LIN {X -0.265,Y -656.677,Z 1261.343,A 0.000,B 0.000,C 90.000,E1 97.757} C_DIS
LIN {X -0.061,Y -653.194,Z 1261.340,A 0.000,B 0.000,C 90.000,E1 97.125} C_DIS
LIN {X 0.226,Y -650.001,Z 1261.337,A 0.000,B 0.000,C 90.000,E1 96.606} C_DIS
LIN {X -0.200,Y -645.461,Z 1261.333,A 0.000,B 0.000,C 90.000,E1 96.024} C_DIS
LIN {X 0.088,Y -642.536,Z 1261.331,A 0.000,B 0.000,C 90.000,E1 95.625} C_DIS
LIN {X 0.172,Y -637.015,Z 1261.328,A 0.000,B 0.000,C 90.000,E1 94.992} C_DIS
LIN {X 0.261,Y -630.867,Z 1261.324,A 0.000,B 0.000,C 90.000,E1 94.359} C_DIS
LIN {X -0.014,Y -625.710,Z 1261.322,A 0.000,B 0.000,C 90.000,E1 93.898} C_DIS
LIN {X -0.161,Y -618.882,Z 1261.318,A 0.000,B 0.000,C 90.000,E1 93.326} C_DIS
LIN {X -0.104,Y -614.516,Z 1261.317,A 0.000,B 0.000,C 90.000,E1 92.980} C_DIS
LIN {X 0.202,Y -608.733,Z 1261.314,A 0.000,B 0.000,C 90.000,E1 92.522} C_DIS
LIN {X 0.170,Y -601.165,Z 1261.311,A 0.000,B 0.000,C 90.000,E1 92.007} C_DIS
LIN {X 0.030,Y -596.550,Z 1261.310,A 0.000,B 0.000,C 90.000,E1 91.718} C_DIS
LIN {X 0.285,Y -589.902,Z 1261.307,A 0.000,B 0.000,C 90.000,E1 91.318} C_DIS
LIN {X -0.224,Y -582.805,Z 1261.306,A 0.000,B 0.000,C 90.000,E1 91.031} C_DIS
LIN {X 0.245,Y -572.407,Z 1261.303,A 0.000,B 0.000,C 90.000,E1 90.573} C_DIS
LIN {X -0.107,Y -571.604,Z 1261.303,A 0.000,B 0.000,C 90.000,E1 90.573} C_DIS
LIN {X -0.091,Y -568.535,Z 1261.302,A 0.000,B 0.000,C 90.000,E1 90.286} C_DIS
LIN {X -0.129,Y -568.514,Z 1261.302,A 0.000,B 0.000,C 90.000,E1 90.286} C_DIS
LIN {X 0.130,Y -568.042,Z 1261.300,A 0.000,B 0.000,C 90.000,E1 90.057} C_DIS
LIN {X -0.091,Y -567.850,Z 1261.300,A 0.000,B 0.000,C 90.000,E1 89.943} C_DIS
LIN {X -0.185,Y -567.751,Z 1261.297,A 0.000,B 0.000,C 90.000,E1 89.542} C_DIS
LIN {X 0.077,Y -570.055,Z 1261.281,A 0.000,B 0.000,C 90.000,E1 86.502} C_DIS
LIN {X -0.107,Y -571.867,Z 1261.270,A 0.000,B 0.000,C 90.000,E1 84.609} C_DIS
LIN {X 0.116,Y -573.308,Z 1261.262,A 0.000,B 0.000,C 90.000,E1 83.223} C_DIS
LIN {X 0.172,Y -574.522,Z 1261.256,A 0.000,B 0.000,C 90.000,E1 82.129} C_DIS
LIN {X -0.043,Y -575.996,Z 1261.249,A 0.000,B 0.000,C 90.000,E1 80.792} C_DIS
LIN {X -0.226,Y -577.274,Z 1261.241,A 0.000,B 0.000,C 90.000,E1 79.454} C_DIS
LIN {X -0.056,Y -578.563,Z 1261.232,A 0.000,B 0.000,C 90.000,E1 77.813} C_DIS
LIN {X -0.082,Y -579.546,Z 1261.225,A 0.000,B 0.000,C 90.000,E1 76.464} C_DIS
LIN {X 0.266,Y -580.700,Z 1261.216,A 0.000,B 0.000,C 90.000,E1 74.810} C_DIS
LIN {X 0.229,Y -581.613,Z 1261.207,A 0.000,B 0.000,C 90.000,E1 73.196} C_DIS
LIN {X 0.207,Y -582.610,Z 1261.198,A 0.000,B 0.000,C 90.000,E1 71.583} C_DIS
LIN {X 0.171,Y -583.419,Z 1261.190,A 0.000,B 0.000,C 90.000,E1 70.242} C_DIS
LIN {X 0.075,Y -584.653,Z 1261.178,A 0.000,B 0.000,C 90.000,E1 68.103} C_DIS
LIN {X 0.210,Y -586.714,Z 1261.164,A 0.000,B 0.000,C 90.000,E1 65.409} C_DIS
LIN {X 0.165,Y -587.802,Z 1261.156,A 0.000,B 0.000,C 90.000,E1 64.076} C_DIS
LIN {X -0.196,Y -589.681,Z 1261.144,A 0.000,B 0.000,C 90.000,E1 61.975} C_DIS
LIN {X 0.244,Y -591.320,Z 1261.135,A 0.000,B 0.000,C 90.000,E1 60.333} C_DIS
LIN {X 0.314,Y -592.676,Z 1261.128,A 0.000,B 0.000,C 90.000,E1 58.997} C_DIS
LIN {X -0.306,Y -593.785,Z 1261.122,A 0.000,B 0.000,C 90.000,E1 57.995} C_DIS
LIN {X 0.122,Y -595.104,Z 1261.115,A 0.000,B 0.000,C 90.000,E1 56.628} C_DIS
LIN {X -0.148,Y -596.182,Z 1261.109,A 0.000,B 0.000,C 90.000,E1 55.595} C_DIS
LIN {X -0.177,Y -597.375,Z 1261.101,A 0.000,B 0.000,C 90.000,E1 54.276} C_DIS
LIN {X 0.159,Y -598.492,Z 1261.094,A 0.000,B 0.000,C 90.000,E1 52.924} C_DIS
LIN {X -0.190,Y -599.747,Z 1261.085,A 0.000,B 0.000,C 90.000,E1 51.376} C_DIS
LIN {X 0.312,Y -600.507,Z 1261.079,A 0.000,B 0.000,C 90.000,E1 50.275} C_DIS
LIN {X -0.269,Y -600.857,Z 1261.075,A 0.000,B 0.000,C 90.000,E1 49.542} C_DIS
LIN {X 0.418,Y -601.419,Z 1261.068,A 0.000,B 0.000,C 90.000,E1 48.162} C_DIS
LIN {X -0.177,Y -601.855,Z 1261.061,A 0.000,B 0.000,C 90.000,E1 46.905} C_DIS
LIN {X 0.087,Y -602.192,Z 1261.053,A 0.000,B 0.000,C 90.000,E1 45.567} C_DIS
LIN {X 0.126,Y -602.208,Z 1261.047,A 0.000,B 0.000,C 90.000,E1 44.514} C_DIS
LIN {X 0.162,Y -602.014,Z 1261.042,A 0.000,B 0.000,C 90.000,E1 43.461} C_DIS
LIN {X -0.223,Y -601.693,Z 1261.036,A 0.000,B 0.000,C 90.000,E1 42.447} C_DIS
LIN {X -0.131,Y -601.087,Z 1261.027,A 0.000,B 0.000,C 90.000,E1 40.862} C_DIS
LIN {X -0.073,Y -600.537,Z 1261.021,A 0.000,B 0.000,C 90.000,E1 39.806} C_DIS
LIN {X 0.214,Y -599.664,Z 1261.014,A 0.000,B 0.000,C 90.000,E1 38.463} C_DIS
LIN {X -0.133,Y -598.800,Z 1261.008,A 0.000,B 0.000,C 90.000,E1 37.443} C_DIS
LIN {X 0.347,Y -598.249,Z 1261.005,A 0.000,B 0.000,C 90.000,E1 36.870} C_DIS
LIN {X -0.143,Y -596.548,Z 1260.998,A 0.000,B 0.000,C 90.000,E1 35.598} C_DIS
LIN {X -0.059,Y -594.926,Z 1260.992,A 0.000,B 0.000,C 90.000,E1 34.532} C_DIS
LIN {X -0.126,Y -592.297,Z 1260.984,A 0.000,B 0.000,C 90.000,E1 33.214} C_DIS
LIN {X -0.147,Y -590.449,Z 1260.980,A 0.000,B 0.000,C 90.000,E1 32.418} C_DIS
LIN {X 0.012,Y -587.470,Z 1260.974,A 0.000,B 0.000,C 90.000,E1 31.337} C_DIS
LIN {X -0.048,Y -584.780,Z 1260.970,A 0.000,B 0.000,C 90.000,E1 30.541} C_DIS
LIN {X -0.005,Y -582.817,Z 1260.967,A 0.000,B 0.000,C 90.000,E1 30.001} C_DIS
LIN {X 0.020,Y -580.621,Z 1260.964,A 0.000,B 0.000,C 90.000,E1 29.461} C_DIS
LIN {X -0.324,Y -577.596,Z 1260.960,A 0.000,B 0.000,C 90.000,E1 28.821} C_DIS
LIN {X -0.066,Y -572.874,Z 1260.955,A 0.000,B 0.000,C 90.000,E1 27.847} C_DIS
LIN {X 0.298,Y -569.137,Z 1260.951,A 0.000,B 0.000,C 90.000,E1 27.129} C_DIS
LIN {X -0.137,Y -564.947,Z 1260.947,A 0.000,B 0.000,C 90.000,E1 26.488} C_DIS
LIN {X -0.196,Y -559.579,Z 1260.943,A 0.000,B 0.000,C 90.000,E1 25.668} C_DIS
LIN {X 0.139,Y -555.677,Z 1260.939,A 0.000,B 0.000,C 90.000,E1 25.079} C_DIS
LIN {X 0.092,Y -550.432,Z 1260.936,A 0.000,B 0.000,C 90.000,E1 24.387} C_DIS
LIN {X -0.082,Y -542.758,Z 1260.930,A 0.000,B 0.000,C 90.000,E1 23.462} C_DIS
LIN {X -0.055,Y -536.736,Z 1260.927,A 0.000,B 0.000,C 90.000,E1 22.770} C_DIS
LIN {X -0.017,Y -530.447,Z 1260.923,A 0.000,B 0.000,C 90.000,E1 22.078} C_DIS
LIN {X -0.265,Y -523.824,Z 1260.919,A 0.000,B 0.000,C 90.000,E1 21.408} C_DIS
LIN {X -0.178,Y -514.447,Z 1260.913,A 0.000,B 0.000,C 90.000,E1 20.429} C_DIS
LIN {X 0.084,Y -507.610,Z 1260.910,A 0.000,B 0.000,C 90.000,E1 19.704} C_DIS
LIN {X -0.194,Y -495.124,Z 1260.903,A 0.000,B 0.000,C 90.000,E1 18.544} C_DIS
LIN {X 0.160,Y -485.220,Z 1260.898,A 0.000,B 0.000,C 90.000,E1 17.583} C_DIS
LIN {X 0.219,Y -477.861,Z 1260.894,A 0.000,B 0.000,C 90.000,E1 16.913} C_DIS
LIN {X -0.094,Y -463.272,Z 1260.887,A 0.000,B 0.000,C 90.000,E1 15.662} C_DIS
LIN {X 0.064,Y -444.094,Z 1260.877,A 0.000,B 0.000,C 90.000,E1 13.883} C_DIS
LIN {X -0.057,Y -423.794,Z 1260.866,A 0.000,B 0.000,C 90.000,E1 11.883} C_DIS
LIN {X 0.104,Y -406.795,Z 1260.856,A 0.000,B 0.000,C 90.000,E1 10.018} C_DIS
LIN {X 0.018,Y -400.189,Z 1260.852,A 0.000,B 0.000,C 90.000,E1 9.265} C_DIS
LIN {X 0.095,Y -397.509,Z 1260.850,A 0.000,B 0.000,C 90.000,E1 8.916} C_DIS
LIN {X -0.096,Y -394.827,Z 1260.847,A 0.000,B 0.000,C 90.000,E1 8.511} C_DIS
LIN {X 0.117,Y -394.566,Z 1260.847,A 0.000,B 0.000,C 90.000,E1 8.398} C_DIS
LIN {X 0.080,Y -394.582,Z 1260.847,A 0.000,B 0.000,C 90.000,E1 8.398} C_DIS
LIN {X -0.041,Y -395.842,Z 1260.845,A 0.000,B 0.000,C 90.000,E1 8.106} C_DIS
LIN {X 0.133,Y -396.455,Z 1260.845,A 0.000,B 0.000,C 90.000,E1 7.992} C_DIS
LIN {X -0.104,Y -400.631,Z 1260.842,A 0.000,B 0.000,C 90.000,E1 7.644} C_DIS
LIN {X -0.068,Y -404.555,Z 1260.841,A 0.000,B 0.000,C 90.000,E1 7.352} C_DIS
LIN {X -0.113,Y -416.122,Z 1260.837,A 0.000,B 0.000,C 90.000,E1 6.606} C_DIS
LIN {X 0.122,Y -423.823,Z 1260.834,A 0.000,B 0.000,C 90.000,E1 6.030} C_DIS
LIN {X -0.032,Y -433.217,Z 1260.830,A 0.000,B 0.000,C 90.000,E1 5.334} C_DIS
LIN {X 0.061,Y -442.531,Z 1260.826,A 0.000,B 0.000,C 90.000,E1 4.588} C_DIS
LIN {X -0.199,Y -454.787,Z 1260.820,A 0.000,B 0.000,C 90.000,E1 3.612} C_DIS
LIN {X 0.082,Y -460.469,Z 1260.817,A 0.000,B 0.000,C 90.000,E1 3.094} C_DIS
LIN {X -0.145,Y -467.790,Z 1260.814,A 0.000,B 0.000,C 90.000,E1 2.465} C_DIS
LIN {X 0.030,Y -473.481,Z 1260.811,A 0.000,B 0.000,C 90.000,E1 1.892} C_DIS
LIN {X 0.043,Y -479.042,Z 1260.807,A 0.000,B 0.000,C 90.000,E1 1.318} C_DIS
LIN {X 0.128,Y -485.659,Z 1260.803,A 0.000,B 0.000,C 90.000,E1 0.573} C_DIS
LIN {X 0.000,Y -490.538,Z 1260.800,A 0.000,B 0.000,C 90.000,E1 360.000} C_DIS
LIN {X 0.030,Y -494.624,Z 1260.797,A 0.000,B 0.000,C 90.000,E1 359.484} C_DIS
LIN {X -0.074,Y -500.095,Z 1260.793,A 0.000,B 0.000,C 90.000,E1 358.740} C_DIS
LIN {X 0.081,Y -506.104,Z 1260.788,A 0.000,B 0.000,C 90.000,E1 357.822} C_DIS
LIN {X -0.128,Y -509.961,Z 1260.785,A 0.000,B 0.000,C 90.000,E1 357.249} C_DIS
LIN {X 0.144,Y -515.226,Z 1260.780,A 0.000,B 0.000,C 90.000,E1 356.331} C_DIS
LIN {X 0.029,Y -518.532,Z 1260.776,A 0.000,B 0.000,C 90.000,E1 355.755} C_DIS
LIN {X 0.169,Y -522.370,Z 1260.772,A 0.000,B 0.000,C 90.000,E1 355.008} C_DIS
LIN {X 0.108,Y -525.211,Z 1260.769,A 0.000,B 0.000,C 90.000,E1 354.432} C_DIS
LIN {X -0.197,Y -529.795,Z 1260.764,A 0.000,B 0.000,C 90.000,E1 353.451} C_DIS
LIN {X 0.040,Y -532.781,Z 1260.760,A 0.000,B 0.000,C 90.000,E1 352.704} C_DIS
LIN {X 0.090,Y -535.985,Z 1260.755,A 0.000,B 0.000,C 90.000,E1 351.837} C_DIS
LIN {X 0.236,Y -539.866,Z 1260.748,A 0.000,B 0.000,C 90.000,E1 350.679} C_DIS
LIN {X -0.081,Y -542.422,Z 1260.744,A 0.000,B 0.000,C 90.000,E1 349.859} C_DIS
LIN {X 0.152,Y -545.579,Z 1260.737,A 0.000,B 0.000,C 90.000,E1 348.701} C_DIS
LIN {X -0.006,Y -548.332,Z 1260.731,A 0.000,B 0.000,C 90.000,E1 347.589} C_DIS
LIN {X 0.108,Y -551.388,Z 1260.723,A 0.000,B 0.000,C 90.000,E1 346.172} C_DIS
LIN {X 0.048,Y -552.970,Z 1260.719,A 0.000,B 0.000,C 90.000,E1 345.338} C_DIS
LIN {X 0.129,Y -554.793,Z 1260.712,A 0.000,B 0.000,C 90.000,E1 344.212} C_DIS
LIN {X 0.108,Y -556.002,Z 1260.708,A 0.000,B 0.000,C 90.000,E1 343.378} C_DIS
LIN {X -0.315,Y -557.406,Z 1260.702,A 0.000,B 0.000,C 90.000,E1 342.308} C_DIS
LIN {X -0.143,Y -558.149,Z 1260.697,A 0.000,B 0.000,C 90.000,E1 341.456} C_DIS
LIN {X -0.258,Y -558.518,Z 1260.694,A 0.000,B 0.000,C 90.000,E1 340.913} C_DIS
LIN {X 0.234,Y -558.939,Z 1260.688,A 0.000,B 0.000,C 90.000,E1 339.752} C_DIS
LIN {X -0.096,Y -558.797,Z 1260.683,A 0.000,B 0.000,C 90.000,E1 338.954} C_DIS
LIN {X 0.090,Y -558.371,Z 1260.678,A 0.000,B 0.000,C 90.000,E1 338.103} C_DIS
LIN {X 0.048,Y -557.325,Z 1260.672,A 0.000,B 0.000,C 90.000,E1 336.997} C_DIS
LIN {X 0.127,Y -556.592,Z 1260.669,A 0.000,B 0.000,C 90.000,E1 336.433} C_DIS
LIN {X -0.014,Y -555.313,Z 1260.665,A 0.000,B 0.000,C 90.000,E1 335.613} C_DIS
LIN {X 0.110,Y -553.121,Z 1260.658,A 0.000,B 0.000,C 90.000,E1 334.485} C_DIS
LIN {X 0.173,Y -551.209,Z 1260.654,A 0.000,B 0.000,C 90.000,E1 333.640} C_DIS
LIN {X -0.056,Y -550.332,Z 1260.652,A 0.000,B 0.000,C 90.000,E1 333.384} C_DIS
LIN {X -0.029,Y -548.896,Z 1260.649,A 0.000,B 0.000,C 90.000,E1 332.820} C_DIS
LIN {X -0.007,Y -545.973,Z 1260.644,A 0.000,B 0.000,C 90.000,E1 331.975} C_DIS
LIN {X 0.008,Y -544.925,Z 1260.643,A 0.000,B 0.000,C 90.000,E1 331.691} C_DIS
LIN {X -0.139,Y -540.543,Z 1260.637,A 0.000,B 0.000,C 90.000,E1 330.717} C_DIS
LIN {X 0.064,Y -537.784,Z 1260.634,A 0.000,B 0.000,C 90.000,E1 330.127} C_DIS
LIN {X 0.102,Y -533.880,Z 1260.630,A 0.000,B 0.000,C 90.000,E1 329.410} C_DIS
LIN {X 0.221,Y -528.471,Z 1260.625,A 0.000,B 0.000,C 90.000,E1 328.535} C_DIS
LIN {X 0.117,Y -521.904,Z 1260.620,A 0.000,B 0.000,C 90.000,E1 327.533} C_DIS
LIN {X -0.332,Y -516.216,Z 1260.615,A 0.000,B 0.000,C 90.000,E1 326.707} C_DIS
LIN {X 0.063,Y -511.937,Z 1260.611,A 0.000,B 0.000,C 90.000,E1 325.928} C_DIS
LIN {X 0.029,Y -509.020,Z 1260.608,A 0.000,B 0.000,C 90.000,E1 325.341} C_DIS
LIN {X -0.058,Y -506.129,Z 1260.603,A 0.000,B 0.000,C 90.000,E1 324.609} C_DIS
LIN {X 0.092,Y -503.747,Z 1260.598,A 0.000,B 0.000,C 90.000,E1 323.623} C_DIS
LIN {X -0.235,Y -502.415,Z 1260.593,A 0.000,B 0.000,C 90.000,E1 322.763} C_DIS
LIN {X 0.127,Y -501.900,Z 1260.588,A 0.000,B 0.000,C 90.000,E1 321.823} C_DIS
LIN {X -0.018,Y -502.220,Z 1260.568,A 0.000,B 0.000,C 90.000,E1 318.243} C_DIS
LIN {X -0.004,Y -502.565,Z 1260.560,A 0.000,B 0.000,C 90.000,E1 316.743} C_DIS
LIN {X -0.040,Y -503.090,Z 1260.546,A 0.000,B 0.000,C 90.000,E1 314.352} C_DIS
LIN {X -0.009,Y -503.410,Z 1260.538,A 0.000,B 0.000,C 90.000,E1 312.852} C_DIS
LIN {X 0.021,Y -503.703,Z 1260.530,A 0.000,B 0.000,C 90.000,E1 311.353} C_DIS
LIN {X -0.018,Y -503.979,Z 1260.520,A 0.000,B 0.000,C 90.000,E1 309.564} C_DIS
LIN {X 0.127,Y -504.577,Z 1260.507,A 0.000,B 0.000,C 90.000,E1 307.156} C_DIS
LIN {X -0.214,Y -504.865,Z 1260.495,A 0.000,B 0.000,C 90.000,E1 305.105} C_DIS
LIN {X 0.080,Y -504.967,Z 1260.487,A 0.000,B 0.000,C 90.000,E1 303.579} C_DIS
LIN {X 0.098,Y -504.986,Z 1260.478,A 0.000,B 0.000,C 90.000,E1 302.084} C_DIS
LIN {X -0.267,Y -504.796,Z 1260.468,A 0.000,B 0.000,C 90.000,E1 300.335} C_DIS
LIN {X -0.144,Y -504.676,Z 1260.457,A 0.000,B 0.000,C 90.000,E1 298.231} C_DIS
LIN {X -0.117,Y -504.328,Z 1260.442,A 0.000,B 0.000,C 90.000,E1 295.540} C_DIS
LIN {X 0.054,Y -504.283,Z 1260.434,A 0.000,B 0.000,C 90.000,E1 294.027} C_DIS
LIN {X 0.048,Y -504.109,Z 1260.429,A 0.000,B 0.000,C 90.000,E1 293.131} C_DIS
LIN {X -0.082,Y -503.684,Z 1260.422,A 0.000,B 0.000,C 90.000,E1 291.950} C_DIS
LIN {X 0.066,Y -503.051,Z 1260.415,A 0.000,B 0.000,C 90.000,E1 290.737} C_DIS
LIN {X -0.165,Y -502.280,Z 1260.410,A 0.000,B 0.000,C 90.000,E1 289.866} C_DIS
LIN {X -0.036,Y -501.188,Z 1260.404,A 0.000,B 0.000,C 90.000,E1 288.652} C_DIS
LIN {X -0.079,Y -499.904,Z 1260.397,A 0.000,B 0.000,C 90.000,E1 287.457} C_DIS
LIN {X -0.048,Y -498.664,Z 1260.392,A 0.000,B 0.000,C 90.000,E1 286.551} C_DIS
LIN {X -0.085,Y -497.613,Z 1260.389,A 0.000,B 0.000,C 90.000,E1 285.953} C_DIS
LIN {X -0.261,Y -496.258,Z 1260.385,A 0.000,B 0.000,C 90.000,E1 285.371} C_DIS
LIN {X 0.118,Y -487.594,Z 1260.362,A 0.000,B 0.000,C 90.000,E1 281.074} C_DIS
LIN {X -0.118,Y -480.717,Z 1260.331,A 0.000,B 0.000,C 90.000,E1 275.568} C_DIS
LIN {X -0.123,Y -482.447,Z 1260.260,A 0.000,B 0.000,C 90.000,E1 262.875} C_DIS
LIN {X 0.009,Y -482.831,Z 1260.257,A 0.000,B 0.000,C 90.000,E1 262.243} C_DIS
LIN {X 0.210,Y -482.953,Z 1260.254,A 0.000,B 0.000,C 90.000,E1 261.602} C_DIS
LIN {X 0.068,Y -482.790,Z 1260.247,A 0.000,B 0.000,C 90.000,E1 260.387} C_DIS
LIN {X 0.139,Y -482.456,Z 1260.242,A 0.000,B 0.000,C 90.000,E1 259.454} C_DIS
LIN {X 0.124,Y -481.566,Z 1260.230,A 0.000,B 0.000,C 90.000,E1 257.297} C_DIS
LIN {X -0.183,Y -480.413,Z 1260.218,A 0.000,B 0.000,C 90.000,E1 255.172} C_DIS
LIN {X -0.065,Y -479.771,Z 1260.211,A 0.000,B 0.000,C 90.000,E1 253.921} C_DIS
LIN {X 0.025,Y -478.813,Z 1260.202,A 0.000,B 0.000,C 90.000,E1 252.362} C_DIS
LIN {X 0.072,Y -477.835,Z 1260.192,A 0.000,B 0.000,C 90.000,E1 250.496} C_DIS
LIN {X -0.028,Y -476.919,Z 1260.181,A 0.000,B 0.000,C 90.000,E1 248.646} C_DIS
LIN {X -0.142,Y -475.873,Z 1260.171,A 0.000,B 0.000,C 90.000,E1 246.794} C_DIS
LIN {X -0.104,Y -474.678,Z 1260.161,A 0.000,B 0.000,C 90.000,E1 244.921} C_DIS
LIN {X 0.173,Y -473.883,Z 1260.154,A 0.000,B 0.000,C 90.000,E1 243.640} C_DIS
LIN {X -0.146,Y -472.223,Z 1260.140,A 0.000,B 0.000,C 90.000,E1 241.179} C_DIS
LIN {X 0.008,Y -470.952,Z 1260.129,A 0.000,B 0.000,C 90.000,E1 239.282} C_DIS
LIN {X 0.045,Y -469.719,Z 1260.121,A 0.000,B 0.000,C 90.000,E1 237.709} C_DIS
LIN {X -0.009,Y -467.986,Z 1260.109,A 0.000,B 0.000,C 90.000,E1 235.515} C_DIS
LIN {X -0.051,Y -466.158,Z 1260.093,A 0.000,B 0.000,C 90.000,E1 232.683} C_DIS
LIN {X -0.012,Y -464.970,Z 1260.079,A 0.000,B 0.000,C 90.000,E1 230.150} C_DIS
LIN {X 0.061,Y -464.161,Z 1260.068,A 0.000,B 0.000,C 90.000,E1 228.243} C_DIS
LIN {X -0.137,Y -463.956,Z 1260.065,A 0.000,B 0.000,C 90.000,E1 227.634} C_DIS
LIN {X -0.058,Y -462.871,Z 1260.052,A 0.000,B 0.000,C 90.000,E1 225.405} C_DIS
LIN {X -0.117,Y -461.664,Z 1260.022,A 0.000,B 0.000,C 90.000,E1 220.011} C_DIS
LIN {X -0.162,Y -462.638,Z 1260.006,A 0.000,B 0.000,C 90.000,E1 217.156} C_DIS
LIN {X -0.145,Y -466.336,Z 1259.978,A 0.000,B 0.000,C 90.000,E1 212.084} C_DIS
LIN {X -0.277,Y -469.894,Z 1259.961,A 0.000,B 0.000,C 90.000,E1 208.949} C_DIS
LIN {X 0.150,Y -471.451,Z 1259.954,A 0.000,B 0.000,C 90.000,E1 207.641} C_DIS
LIN {X 0.142,Y -475.404,Z 1259.936,A 0.000,B 0.000,C 90.000,E1 204.515} C_DIS
LIN {X 0.179,Y -478.721,Z 1259.924,A 0.000,B 0.000,C 90.000,E1 202.333} C_DIS
LIN {X -0.046,Y -483.435,Z 1259.909,A 0.000,B 0.000,C 90.000,E1 199.577} C_DIS
LIN {X 0.154,Y -487.674,Z 1259.897,A 0.000,B 0.000,C 90.000,E1 197.402} C_DIS
LIN {X -0.173,Y -491.400,Z 1259.887,A 0.000,B 0.000,C 90.000,E1 195.607} C_DIS
LIN {X -0.054,Y -495.796,Z 1259.875,A 0.000,B 0.000,C 90.000,E1 193.467} C_DIS
LIN {X -0.006,Y -499.129,Z 1259.866,A 0.000,B 0.000,C 90.000,E1 191.951} C_DIS
LIN {X -0.013,Y -503.789,Z 1259.855,A 0.000,B 0.000,C 90.000,E1 189.849} C_DIS
LIN {X 0.060,Y -507.844,Z 1259.845,A 0.000,B 0.000,C 90.000,E1 188.049} C_DIS
LIN {X 0.195,Y -511.311,Z 1259.837,A 0.000,B 0.000,C 90.000,E1 186.549} C_DIS
LIN {X -0.201,Y -515.346,Z 1259.827,A 0.000,B 0.000,C 90.000,E1 184.821} C_DIS
LIN {X -0.009,Y -519.290,Z 1259.817,A 0.000,B 0.000,C 90.000,E1 183.037} C_DIS
LIN {X 0.253,Y -522.510,Z 1259.809,A 0.000,B 0.000,C 90.000,E1 181.547} C_DIS
LIN {X 0.008,Y -526.237,Z 1259.799,A 0.000,B 0.000,C 90.000,E1 179.828} C_DIS
LIN {X -0.136,Y -529.300,Z 1259.791,A 0.000,B 0.000,C 90.000,E1 178.396} C_DIS
LIN {X -0.200,Y -531.648,Z 1259.785,A 0.000,B 0.000,C 90.000,E1 177.249} C_DIS
LIN {X -0.230,Y -533.809,Z 1259.778,A 0.000,B 0.000,C 90.000,E1 176.102} C_DIS
LIN {X -0.198,Y -536.217,Z 1259.770,A 0.000,B 0.000,C 90.000,E1 174.666} C_DIS
LIN {X -0.123,Y -538.075,Z 1259.764,A 0.000,B 0.000,C 90.000,E1 173.514} C_DIS
LIN {X 0.111,Y -540.127,Z 1259.756,A 0.000,B 0.000,C 90.000,E1 172.064} C_DIS
LIN {X -0.301,Y -541.611,Z 1259.750,A 0.000,B 0.000,C 90.000,E1 170.971} C_DIS
LIN {X 0.181,Y -543.612,Z 1259.740,A 0.000,B 0.000,C 90.000,E1 169.218} C_DIS
LIN {X 0.091,Y -544.930,Z 1259.732,A 0.000,B 0.000,C 90.000,E1 167.813} C_DIS
LIN {X 0.019,Y -546.076,Z 1259.725,A 0.000,B 0.000,C 90.000,E1 166.408} C_DIS
LIN {X -0.201,Y -549.910,Z 1259.703,A 0.000,B 0.000,C 90.000,E1 162.489} C_DIS
LIN {X -0.002,Y -552.839,Z 1259.693,A 0.000,B 0.000,C 90.000,E1 160.786} C_DIS
LIN {X -0.015,Y -556.493,Z 1259.686,A 0.000,B 0.000,C 90.000,E1 159.390} C_DIS
LIN {X 0.149,Y -559.254,Z 1259.681,A 0.000,B 0.000,C 90.000,E1 158.539} C_DIS
LIN {X 0.128,Y -563.640,Z 1259.675,A 0.000,B 0.000,C 90.000,E1 157.433} C_DIS
LIN {X -0.214,Y -569.540,Z 1259.668,A 0.000,B 0.000,C 90.000,E1 156.230} C_DIS
LIN {X 0.073,Y -576.345,Z 1259.661,A 0.000,B 0.000,C 90.000,E1 154.973} C_DIS
LIN {X -0.244,Y -586.200,Z 1259.652,A 0.000,B 0.000,C 90.000,E1 153.384} C_DIS
LIN {X 0.049,Y -593.545,Z 1259.645,A 0.000,B 0.000,C 90.000,E1 152.153} C_DIS
LIN {X -0.229,Y -598.352,Z 1259.641,A 0.000,B 0.000,C 90.000,E1 151.385} C_DIS
LIN {X -0.210,Y -603.692,Z 1259.636,A 0.000,B 0.000,C 90.000,E1 150.461} C_DIS
LIN {X -0.176,Y -610.322,Z 1259.629,A 0.000,B 0.000,C 90.000,E1 149.282} C_DIS
LIN {X 0.021,Y -613.829,Z 1259.626,A 0.000,B 0.000,C 90.000,E1 148.614} C_DIS
LIN {X -0.094,Y -616.034,Z 1259.624,A 0.000,B 0.000,C 90.000,E1 148.250} C_DIS
LIN {X 0.157,Y -619.447,Z 1259.620,A 0.000,B 0.000,C 90.000,E1 147.582} C_DIS
LIN {X -0.092,Y -623.396,Z 1259.616,A 0.000,B 0.000,C 90.000,E1 146.834} C_DIS
LIN {X 0.039,Y -627.776,Z 1259.611,A 0.000,B 0.000,C 90.000,E1 145.928} C_DIS
LIN {X -0.138,Y -631.968,Z 1259.606,A 0.000,B 0.000,C 90.000,E1 145.055} C_DIS
LIN {X -0.058,Y -636.165,Z 1259.600,A 0.000,B 0.000,C 90.000,E1 144.036} C_DIS
LIN {X -0.179,Y -638.178,Z 1259.597,A 0.000,B 0.000,C 90.000,E1 143.543} C_DIS
LIN {X 0.109,Y -640.925,Z 1259.593,A 0.000,B 0.000,C 90.000,E1 142.763} C_DIS
LIN {X -0.073,Y -644.382,Z 1259.588,A 0.000,B 0.000,C 90.000,E1 141.778} C_DIS
LIN {X -0.321,Y -647.528,Z 1259.582,A 0.000,B 0.000,C 90.000,E1 140.803} C_DIS
LIN {X -0.151,Y -651.854,Z 1259.574,A 0.000,B 0.000,C 90.000,E1 139.299} C_DIS
LIN {X -0.343,Y -655.256,Z 1259.567,A 0.000,B 0.000,C 90.000,E1 138.081} C_DIS
LIN {X -0.007,Y -657.892,Z 1259.562,A 0.000,B 0.000,C 90.000,E1 137.067} C_DIS
LIN {X 0.307,Y -662.445,Z 1259.552,A 0.000,B 0.000,C 90.000,E1 135.324} C_DIS
LIN {X 0.251,Y -667.269,Z 1259.542,A 0.000,B 0.000,C 90.000,E1 133.623} C_DIS
LIN {X -0.180,Y -671.448,Z 1259.534,A 0.000,B 0.000,C 90.000,E1 132.204} C_DIS
LIN {X -0.059,Y -674.856,Z 1259.528,A 0.000,B 0.000,C 90.000,E1 130.987} C_DIS
LIN {X 0.257,Y -679.499,Z 1259.518,A 0.000,B 0.000,C 90.000,E1 129.277} C_DIS
LIN {X 0.257,Y -683.823,Z 1259.509,A 0.000,B 0.000,C 90.000,E1 127.604} C_DIS
LIN {X 0.135,Y -686.914,Z 1259.502,A 0.000,B 0.000,C 90.000,E1 126.423} C_DIS
LIN {X 0.199,Y -689.804,Z 1259.496,A 0.000,B 0.000,C 90.000,E1 125.231} C_DIS
LIN {X -0.293,Y -691.896,Z 1259.491,A 0.000,B 0.000,C 90.000,E1 124.326} C_DIS
LIN {X 0.072,Y -694.833,Z 1259.483,A 0.000,B 0.000,C 90.000,E1 122.880} C_DIS
LIN {X -0.130,Y -697.171,Z 1259.476,A 0.000,B 0.000,C 90.000,E1 121.720} C_DIS
LIN {X -0.319,Y -698.917,Z 1259.471,A 0.000,B 0.000,C 90.000,E1 120.797} C_DIS
LIN {X 0.402,Y -701.188,Z 1259.463,A 0.000,B 0.000,C 90.000,E1 119.333} C_DIS
LIN {X -0.132,Y -703.007,Z 1259.455,A 0.000,B 0.000,C 90.000,E1 117.975} C_DIS
LIN {X 0.091,Y -703.742,Z 1259.452,A 0.000,B 0.000,C 90.000,E1 117.257} C_DIS
LIN {X 0.031,Y -704.095,Z 1259.449,A 0.000,B 0.000,C 90.000,E1 116.796} C_DIS
LIN {X 0.229,Y -704.412,Z 1259.444,A 0.000,B 0.000,C 90.000,E1 115.848} C_DIS
LIN {X 0.151,Y -704.194,Z 1259.440,A 0.000,B 0.000,C 90.000,E1 115.155} C_DIS
LIN {X -0.214,Y -703.901,Z 1259.437,A 0.000,B 0.000,C 90.000,E1 114.719} C_DIS
LIN {X 0.354,Y -703.119,Z 1259.435,A 0.000,B 0.000,C 90.000,E1 114.207} C_DIS
LIN {X -0.007,Y -702.651,Z 1259.433,A 0.000,B 0.000,C 90.000,E1 114.003} C_DIS
LIN {X 0.263,Y -700.844,Z 1259.431,A 0.000,B 0.000,C 90.000,E1 113.515} C_DIS
LIN {X -0.386,Y -699.622,Z 1259.430,A 0.000,B 0.000,C 90.000,E1 113.334} C_DIS
LIN {X 0.142,Y -695.434,Z 1259.427,A 0.000,B 0.000,C 90.000,E1 112.823} C_DIS
LIN {X -0.001,Y -694.117,Z 1259.426,A 0.000,B 0.000,C 90.000,E1 112.717} C_DIS
LIN {X 0.125,Y -691.987,Z 1259.426,A 0.000,B 0.000,C 90.000,E1 112.589} C_DIS
LIN {X -0.373,Y -687.577,Z 1259.425,A 0.000,B 0.000,C 90.000,E1 112.461} C_DIS
LIN {X -0.239,Y -684.991,Z 1259.424,A 0.000,B 0.000,C 90.000,E1 112.386} C_DIS
LIN {X -0.088,Y -678.907,Z 1259.424,A 0.000,B 0.000,C 90.000,E1 112.259} C_DIS
LIN {X 0.303,Y -677.481,Z 1259.424,A 0.000,B 0.000,C 90.000,E1 112.206} C_DIS
LIN {X 0.067,Y -670.824,Z 1259.423,A 0.000,B 0.000,C 90.000,E1 112.206} C_DIS
LIN {X 0.002,Y -630.925,Z 1259.423,A 0.000,B 0.000,C 90.000,E1 112.206} C_DIS
LIN {X -0.280,Y -628.820,Z 1259.423,A 0.000,B 0.000,C 90.000,E1 112.153} C_DIS
LIN {X -0.322,Y -628.742,Z 1259.423,A 0.000,B 0.000,C 90.000,E1 112.153} C_DIS
LIN {X -0.217,Y -627.629,Z 1259.422,A 0.000,B 0.000,C 90.000,E1 112.025} C_DIS
LIN {X -0.261,Y -627.622,Z 1259.422,A 0.000,B 0.000,C 90.000,E1 112.025} C_DIS
LIN {X -0.288,Y -627.547,Z 1259.422,A 0.000,B 0.000,C 90.000,E1 111.897} C_DIS
LIN {X 0.203,Y -629.498,Z 1259.419,A 0.000,B 0.000,C 90.000,E1 111.408} C_DIS
LIN {X -0.014,Y -637.304,Z 1259.412,A 0.000,B 0.000,C 90.000,E1 110.174} C_DIS
LIN {X 0.281,Y -642.273,Z 1259.407,A 0.000,B 0.000,C 90.000,E1 109.268} C_DIS
LIN {X 0.005,Y -646.027,Z 1259.403,A 0.000,B 0.000,C 90.000,E1 108.544} C_DIS
LIN {X 0.299,Y -651.970,Z 1259.396,A 0.000,B 0.000,C 90.000,E1 107.275} C_DIS
LIN {X 0.105,Y -655.337,Z 1259.392,A 0.000,B 0.000,C 90.000,E1 106.551} C_DIS
LIN {X -0.246,Y -658.439,Z 1259.388,A 0.000,B 0.000,C 90.000,E1 105.843} C_DIS
LIN {X 0.176,Y -660.197,Z 1259.385,A 0.000,B 0.000,C 90.000,E1 105.315} C_DIS
LIN {X 0.050,Y -662.443,Z 1259.381,A 0.000,B 0.000,C 90.000,E1 104.592} C_DIS
LIN {X -0.137,Y -663.682,Z 1259.378,A 0.000,B 0.000,C 90.000,E1 104.120} C_DIS
LIN {X 0.242,Y -665.096,Z 1259.374,A 0.000,B 0.000,C 90.000,E1 103.355} C_DIS
LIN {X 0.072,Y -665.681,Z 1259.372,A 0.000,B 0.000,C 90.000,E1 102.883} C_DIS
LIN {X -0.178,Y -666.041,Z 1259.368,A 0.000,B 0.000,C 90.000,E1 102.175} C_DIS
LIN {X 0.170,Y -666.075,Z 1259.365,A 0.000,B 0.000,C 90.000,E1 101.658} C_DIS
LIN {X -0.081,Y -665.492,Z 1259.361,A 0.000,B 0.000,C 90.000,E1 100.950} C_DIS
LIN {X 0.277,Y -664.870,Z 1259.358,A 0.000,B 0.000,C 90.000,E1 100.433} C_DIS
LIN {X 0.098,Y -663.918,Z 1259.355,A 0.000,B 0.000,C 90.000,E1 99.962} C_DIS
LIN {X -0.201,Y -662.750,Z 1259.353,A 0.000,B 0.000,C 90.000,E1 99.500} C_DIS
LIN {X 0.253,Y -661.209,Z 1259.350,A 0.000,B 0.000,C 90.000,E1 98.973} C_DIS
LIN {X -0.060,Y -659.244,Z 1259.347,A 0.000,B 0.000,C 90.000,E1 98.511} C_DIS
LIN {X 0.270,Y -656.951,Z 1259.345,A 0.000,B 0.000,C 90.000,E1 97.992} C_DIS
LIN {X 0.043,Y -655.050,Z 1259.343,A 0.000,B 0.000,C 90.000,E1 97.644} C_DIS
LIN {X -0.304,Y -652.235,Z 1259.340,A 0.000,B 0.000,C 90.000,E1 97.182} C_DIS
LIN {X -0.023,Y -649.035,Z 1259.337,A 0.000,B 0.000,C 90.000,E1 96.663} C_DIS
LIN {X 0.119,Y -644.459,Z 1259.334,A 0.000,B 0.000,C 90.000,E1 96.030} C_DIS
LIN {X -0.293,Y -640.461,Z 1259.331,A 0.000,B 0.000,C 90.000,E1 95.568} C_DIS
LIN {X -0.093,Y -635.996,Z 1259.328,A 0.000,B 0.000,C 90.000,E1 95.049} C_DIS
LIN {X 0.127,Y -631.110,Z 1259.325,A 0.000,B 0.000,C 90.000,E1 94.531} C_DIS
LIN {X -0.276,Y -624.593,Z 1259.322,A 0.000,B 0.000,C 90.000,E1 93.955} C_DIS
LIN {X 0.234,Y -617.785,Z 1259.319,A 0.000,B 0.000,C 90.000,E1 93.326} C_DIS
LIN {X -0.169,Y -612.014,Z 1259.316,A 0.000,B 0.000,C 90.000,E1 92.922} C_DIS
LIN {X 0.063,Y -607.575,Z 1259.314,A 0.000,B 0.000,C 90.000,E1 92.579} C_DIS
LIN {X -0.083,Y -601.504,Z 1259.312,A 0.000,B 0.000,C 90.000,E1 92.178} C_DIS
LIN {X -0.056,Y -595.258,Z 1259.310,A 0.000,B 0.000,C 90.000,E1 91.776} C_DIS
LIN {X 0.015,Y -590.371,Z 1259.308,A 0.000,B 0.000,C 90.000,E1 91.489} C_DIS
LIN {X 0.292,Y -585.036,Z 1259.307,A 0.000,B 0.000,C 90.000,E1 91.203} C_DIS
LIN {X -0.126,Y -581.531,Z 1259.306,A 0.000,B 0.000,C 90.000,E1 91.088} C_DIS
LIN {X -0.026,Y -573.087,Z 1259.304,A 0.000,B 0.000,C 90.000,E1 90.745} C_DIS
LIN {X 0.058,Y -570.731,Z 1259.304,A 0.000,B 0.000,C 90.000,E1 90.630} C_DIS
LIN {X 0.010,Y -568.377,Z 1259.302,A 0.000,B 0.000,C 90.000,E1 90.401} C_DIS
LIN {X -0.029,Y -568.351,Z 1259.302,A 0.000,B 0.000,C 90.000,E1 90.401} C_DIS
LIN {X 0.025,Y -568.233,Z 1259.302,A 0.000,B 0.000,C 90.000,E1 90.286} C_DIS
LIN {X 0.149,Y -567.683,Z 1259.300,A 0.000,B 0.000,C 90.000,E1 90.000} C_DIS
LIN {X -0.174,Y -567.635,Z 1259.297,A 0.000,B 0.000,C 90.000,E1 89.484} C_DIS
LIN {X -0.193,Y -569.554,Z 1259.283,A 0.000,B 0.000,C 90.000,E1 87.020} C_DIS
LIN {X -0.046,Y -571.855,Z 1259.270,A 0.000,B 0.000,C 90.000,E1 84.546} C_DIS
LIN {X -0.259,Y -573.608,Z 1259.261,A 0.000,B 0.000,C 90.000,E1 82.932} C_DIS
LIN {X 0.003,Y -575.098,Z 1259.253,A 0.000,B 0.000,C 90.000,E1 81.546} C_DIS
LIN {X -0.193,Y -576.488,Z 1259.245,A 0.000,B 0.000,C 90.000,E1 80.208} C_DIS
LIN {X -0.014,Y -577.430,Z 1259.240,A 0.000,B 0.000,C 90.000,E1 79.106} C_DIS
LIN {X -0.189,Y -578.906,Z 1259.229,A 0.000,B 0.000,C 90.000,E1 77.229} C_DIS
LIN {X 0.002,Y -580.017,Z 1259.220,A 0.000,B 0.000,C 90.000,E1 75.589} C_DIS
LIN {X 0.282,Y -580.891,Z 1259.213,A 0.000,B 0.000,C 90.000,E1 74.212} C_DIS
LIN {X -0.089,Y -581.961,Z 1259.202,A 0.000,B 0.000,C 90.000,E1 72.362} C_DIS
LIN {X -0.324,Y -582.823,Z 1259.195,A 0.000,B 0.000,C 90.000,E1 71.040} C_DIS
LIN {X 0.188,Y -583.585,Z 1259.187,A 0.000,B 0.000,C 90.000,E1 69.645} C_DIS
LIN {X -0.240,Y -584.900,Z 1259.175,A 0.000,B 0.000,C 90.000,E1 67.539} C_DIS
LIN {X 0.145,Y -586.617,Z 1259.163,A 0.000,B 0.000,C 90.000,E1 65.357} C_DIS
LIN {X 0.092,Y -587.702,Z 1259.156,A 0.000,B 0.000,C 90.000,E1 64.024} C_DIS
LIN {X -0.004,Y -589.614,Z 1259.144,A 0.000,B 0.000,C 90.000,E1 61.897} C_DIS
LIN {X -0.151,Y -590.717,Z 1259.138,A 0.000,B 0.000,C 90.000,E1 60.845} C_DIS
LIN {X 0.122,Y -592.097,Z 1259.131,A 0.000,B 0.000,C 90.000,E1 59.488} C_DIS
LIN {X -0.308,Y -593.469,Z 1259.123,A 0.000,B 0.000,C 90.000,E1 58.201} C_DIS
LIN {X 0.112,Y -594.780,Z 1259.116,A 0.000,B 0.000,C 90.000,E1 56.834} C_DIS
LIN {X -0.049,Y -596.360,Z 1259.107,A 0.000,B 0.000,C 90.000,E1 55.261} C_DIS
LIN {X -0.333,Y -597.751,Z 1259.098,A 0.000,B 0.000,C 90.000,E1 53.703} C_DIS
LIN {X -0.225,Y -599.005,Z 1259.089,A 0.000,B 0.000,C 90.000,E1 52.110} C_DIS
LIN {X -0.109,Y -599.845,Z 1259.084,A 0.000,B 0.000,C 90.000,E1 51.045} C_DIS
LIN {X 0.145,Y -600.383,Z 1259.079,A 0.000,B 0.000,C 90.000,E1 50.231} C_DIS
LIN {X -0.005,Y -601.174,Z 1259.069,A 0.000,B 0.000,C 90.000,E1 48.405} C_DIS
LIN {X 0.244,Y -601.636,Z 1259.062,A 0.000,B 0.000,C 90.000,E1 47.067} C_DIS
LIN {X 0.300,Y -602.059,Z 1259.053,A 0.000,B 0.000,C 90.000,E1 45.486} C_DIS
LIN {X 0.337,Y -602.025,Z 1259.047,A 0.000,B 0.000,C 90.000,E1 44.433} C_DIS
LIN {X -0.044,Y -601.829,Z 1259.041,A 0.000,B 0.000,C 90.000,E1 43.419} C_DIS
LIN {X -0.018,Y -601.503,Z 1259.035,A 0.000,B 0.000,C 90.000,E1 42.366} C_DIS
LIN {X 0.069,Y -600.923,Z 1259.027,A 0.000,B 0.000,C 90.000,E1 40.782} C_DIS
LIN {X -0.098,Y -600.154,Z 1259.019,A 0.000,B 0.000,C 90.000,E1 39.483} C_DIS
LIN {X 0.030,Y -599.419,Z 1259.014,A 0.000,B 0.000,C 90.000,E1 38.418} C_DIS
LIN {X -0.188,Y -598.797,Z 1259.009,A 0.000,B 0.000,C 90.000,E1 37.649} C_DIS
LIN {X -0.310,Y -597.974,Z 1259.005,A 0.000,B 0.000,C 90.000,E1 36.870} C_DIS
LIN {X -0.203,Y -596.644,Z 1258.999,A 0.000,B 0.000,C 90.000,E1 35.804} C_DIS
LIN {X -0.117,Y -595.053,Z 1258.993,A 0.000,B 0.000,C 90.000,E1 34.739} C_DIS
LIN {X -0.008,Y -594.087,Z 1258.990,A 0.000,B 0.000,C 90.000,E1 34.199} C_DIS
LIN {X -0.295,Y -591.996,Z 1258.984,A 0.000,B 0.000,C 90.000,E1 33.166} C_DIS
LIN {X 0.002,Y -590.048,Z 1258.980,A 0.000,B 0.000,C 90.000,E1 32.339} C_DIS
LIN {X 0.151,Y -587.068,Z 1258.974,A 0.000,B 0.000,C 90.000,E1 31.258} C_DIS
LIN {X 0.208,Y -585.290,Z 1258.971,A 0.000,B 0.000,C 90.000,E1 30.718} C_DIS
LIN {X 0.120,Y -582.288,Z 1258.966,A 0.000,B 0.000,C 90.000,E1 29.922} C_DIS
LIN {X -0.146,Y -580.060,Z 1258.963,A 0.000,B 0.000,C 90.000,E1 29.411} C_DIS
LIN {X -0.212,Y -576.982,Z 1258.960,A 0.000,B 0.000,C 90.000,E1 28.743} C_DIS
LIN {X 0.192,Y -573.629,Z 1258.956,A 0.000,B 0.000,C 90.000,E1 28.025} C_DIS
LIN {X -0.046,Y -571.506,Z 1258.954,A 0.000,B 0.000,C 90.000,E1 27.641} C_DIS
LIN {X 0.129,Y -568.427,Z 1258.951,A 0.000,B 0.000,C 90.000,E1 27.078} C_DIS
LIN {X -0.056,Y -564.206,Z 1258.947,A 0.000,B 0.000,C 90.000,E1 26.411} C_DIS
LIN {X -0.127,Y -558.799,Z 1258.942,A 0.000,B 0.000,C 90.000,E1 25.591} C_DIS
LIN {X -0.144,Y -553.814,Z 1258.938,A 0.000,B 0.000,C 90.000,E1 24.899} C_DIS
LIN {X -0.086,Y -549.503,Z 1258.935,A 0.000,B 0.000,C 90.000,E1 24.335} C_DIS
LIN {X -0.059,Y -544.972,Z 1258.932,A 0.000,B 0.000,C 90.000,E1 23.770} C_DIS
LIN {X -0.065,Y -540.186,Z 1258.929,A 0.000,B 0.000,C 90.000,E1 23.206} C_DIS
LIN {X -0.179,Y -532.770,Z 1258.924,A 0.000,B 0.000,C 90.000,E1 22.386} C_DIS
LIN {X 0.027,Y -526.189,Z 1258.920,A 0.000,B 0.000,C 90.000,E1 21.663} C_DIS
LIN {X -0.251,Y -517.011,Z 1258.915,A 0.000,B 0.000,C 90.000,E1 20.737} C_DIS
LIN {X 0.023,Y -507.685,Z 1258.910,A 0.000,B 0.000,C 90.000,E1 19.758} C_DIS
LIN {X -0.056,Y -494.893,Z 1258.903,A 0.000,B 0.000,C 90.000,E1 18.544} C_DIS
LIN {X -0.015,Y -485.113,Z 1258.898,A 0.000,B 0.000,C 90.000,E1 17.638} C_DIS
LIN {X 0.004,Y -477.925,Z 1258.894,A 0.000,B 0.000,C 90.000,E1 16.985} C_DIS
LIN {X 0.236,Y -463.272,Z 1258.887,A 0.000,B 0.000,C 90.000,E1 15.662} C_DIS
LIN {X 0.059,Y -445.530,Z 1258.878,A 0.000,B 0.000,C 90.000,E1 14.064} C_DIS
LIN {X 0.099,Y -423.688,Z 1258.866,A 0.000,B 0.000,C 90.000,E1 11.895} C_DIS
LIN {X 0.184,Y -406.521,Z 1258.856,A 0.000,B 0.000,C 90.000,E1 10.018} C_DIS
LIN {X -0.192,Y -399.577,Z 1258.851,A 0.000,B 0.000,C 90.000,E1 9.265} C_DIS
LIN {X -0.123,Y -396.959,Z 1258.849,A 0.000,B 0.000,C 90.000,E1 8.916} C_DIS
LIN {X -0.131,Y -394.555,Z 1258.847,A 0.000,B 0.000,C 90.000,E1 8.511} C_DIS
LIN {X -0.166,Y -394.543,Z 1258.847,A 0.000,B 0.000,C 90.000,E1 8.511} C_DIS
LIN {X 0.083,Y -394.507,Z 1258.847,A 0.000,B 0.000,C 90.000,E1 8.454} C_DIS
LIN {X 0.048,Y -394.517,Z 1258.847,A 0.000,B 0.000,C 90.000,E1 8.454} C_DIS
LIN {X -0.022,Y -396.300,Z 1258.845,A 0.000,B 0.000,C 90.000,E1 8.049} C_DIS
LIN {X 0.013,Y -399.956,Z 1258.843,A 0.000,B 0.000,C 90.000,E1 7.701} C_DIS
LIN {X 0.144,Y -405.896,Z 1258.840,A 0.000,B 0.000,C 90.000,E1 7.239} C_DIS
LIN {X 0.028,Y -414.078,Z 1258.837,A 0.000,B 0.000,C 90.000,E1 6.720} C_DIS
LIN {X 0.106,Y -417.454,Z 1258.836,A 0.000,B 0.000,C 90.000,E1 6.486} C_DIS
LIN {X 0.152,Y -425.310,Z 1258.833,A 0.000,B 0.000,C 90.000,E1 5.910} C_DIS
LIN {X -0.076,Y -434.836,Z 1258.829,A 0.000,B 0.000,C 90.000,E1 5.220} C_DIS
LIN {X -0.074,Y -444.121,Z 1258.825,A 0.000,B 0.000,C 90.000,E1 4.473} C_DIS
LIN {X 0.180,Y -454.924,Z 1258.820,A 0.000,B 0.000,C 90.000,E1 3.555} C_DIS
LIN {X 0.232,Y -460.988,Z 1258.817,A 0.000,B 0.000,C 90.000,E1 3.037} C_DIS
LIN {X 0.115,Y -466.930,Z 1258.814,A 0.000,B 0.000,C 90.000,E1 2.522} C_DIS
LIN {X -0.105,Y -472.696,Z 1258.811,A 0.000,B 0.000,C 90.000,E1 2.007} C_DIS
LIN {X -0.223,Y -479.528,Z 1258.807,A 0.000,B 0.000,C 90.000,E1 1.318} C_DIS
LIN {X -0.112,Y -486.146,Z 1258.803,A 0.000,B 0.000,C 90.000,E1 0.573} C_DIS
LIN {X 0.000,Y -490.788,Z 1258.800,A 0.000,B 0.000,C 90.000,E1 360.000} C_DIS
LIN {X 0.031,Y -494.935,Z 1258.797,A 0.000,B 0.000,C 90.000,E1 359.484} C_DIS
LIN {X -0.070,Y -500.410,Z 1258.793,A 0.000,B 0.000,C 90.000,E1 358.740} C_DIS
LIN {X 0.089,Y -506.475,Z 1258.788,A 0.000,B 0.000,C 90.000,E1 357.822} C_DIS
LIN {X -0.117,Y -510.334,Z 1258.785,A 0.000,B 0.000,C 90.000,E1 357.249} C_DIS
LIN {X 0.158,Y -515.638,Z 1258.780,A 0.000,B 0.000,C 90.000,E1 356.331} C_DIS
LIN {X 0.047,Y -518.944,Z 1258.776,A 0.000,B 0.000,C 90.000,E1 355.755} C_DIS
LIN {X 0.191,Y -522.781,Z 1258.772,A 0.000,B 0.000,C 90.000,E1 355.008} C_DIS
LIN {X 0.134,Y -525.642,Z 1258.769,A 0.000,B 0.000,C 90.000,E1 354.432} C_DIS
LIN {X 0.056,Y -529.591,Z 1258.764,A 0.000,B 0.000,C 90.000,E1 353.571} C_DIS
LIN {X 0.075,Y -533.218,Z 1258.760,A 0.000,B 0.000,C 90.000,E1 352.704} C_DIS
LIN {X 0.132,Y -536.407,Z 1258.755,A 0.000,B 0.000,C 90.000,E1 351.837} C_DIS
LIN {X -0.248,Y -540.316,Z 1258.748,A 0.000,B 0.000,C 90.000,E1 350.735} C_DIS
LIN {X -0.027,Y -542.859,Z 1258.744,A 0.000,B 0.000,C 90.000,E1 349.859} C_DIS
LIN {X 0.213,Y -546.026,Z 1258.737,A 0.000,B 0.000,C 90.000,E1 348.701} C_DIS
LIN {X 0.061,Y -548.772,Z 1258.731,A 0.000,B 0.000,C 90.000,E1 347.589} C_DIS
LIN {X 0.073,Y -551.260,Z 1258.725,A 0.000,B 0.000,C 90.000,E1 346.464} C_DIS
LIN {X -0.126,Y -552.951,Z 1258.720,A 0.000,B 0.000,C 90.000,E1 345.644} C_DIS
LIN {X -0.053,Y -554.849,Z 1258.714,A 0.000,B 0.000,C 90.000,E1 344.519} C_DIS
LIN {X 0.202,Y -556.519,Z 1258.708,A 0.000,B 0.000,C 90.000,E1 343.378} C_DIS
LIN {X -0.214,Y -557.947,Z 1258.702,A 0.000,B 0.000,C 90.000,E1 342.308} C_DIS
LIN {X 0.082,Y -558.942,Z 1258.695,A 0.000,B 0.000,C 90.000,E1 341.167} C_DIS
LIN {X 0.047,Y -559.467,Z 1258.689,A 0.000,B 0.000,C 90.000,E1 340.061} C_DIS
LIN {X -0.061,Y -559.588,Z 1258.686,A 0.000,B 0.000,C 90.000,E1 339.518} C_DIS
LIN {X 0.133,Y -559.382,Z 1258.682,A 0.000,B 0.000,C 90.000,E1 338.666} C_DIS
LIN {X 0.011,Y -558.909,Z 1258.677,A 0.000,B 0.000,C 90.000,E1 337.847} C_DIS
LIN {X -0.022,Y -557.804,Z 1258.671,A 0.000,B 0.000,C 90.000,E1 336.741} C_DIS
LIN {X 0.143,Y -556.171,Z 1258.665,A 0.000,B 0.000,C 90.000,E1 335.613} C_DIS
LIN {X -0.072,Y -555.717,Z 1258.663,A 0.000,B 0.000,C 90.000,E1 335.357} C_DIS
LIN {X 0.058,Y -553.421,Z 1258.657,A 0.000,B 0.000,C 90.000,E1 334.229} C_DIS
LIN {X -0.143,Y -552.106,Z 1258.654,A 0.000,B 0.000,C 90.000,E1 333.691} C_DIS
LIN {X 0.159,Y -549.797,Z 1258.649,A 0.000,B 0.000,C 90.000,E1 332.820} C_DIS
LIN {X 0.190,Y -546.933,Z 1258.644,A 0.000,B 0.000,C 90.000,E1 331.975} C_DIS
LIN {X -0.161,Y -544.124,Z 1258.641,A 0.000,B 0.000,C 90.000,E1 331.307} C_DIS
LIN {X -0.056,Y -540.954,Z 1258.637,A 0.000,B 0.000,C 90.000,E1 330.589} C_DIS
LIN {X 0.013,Y -537.325,Z 1258.633,A 0.000,B 0.000,C 90.000,E1 329.871} C_DIS
LIN {X 0.188,Y -534.117,Z 1258.630,A 0.000,B 0.000,C 90.000,E1 329.282} C_DIS
LIN {X 0.277,Y -526.789,Z 1258.623,A 0.000,B 0.000,C 90.000,E1 328.122} C_DIS
LIN {X -0.121,Y -520.989,Z 1258.618,A 0.000,B 0.000,C 90.000,E1 327.296} C_DIS
LIN {X -0.314,Y -514.531,Z 1258.613,A 0.000,B 0.000,C 90.000,E1 326.294} C_DIS
LIN {X -0.153,Y -511.428,Z 1258.609,A 0.000,B 0.000,C 90.000,E1 325.722} C_DIS
LIN {X -0.124,Y -508.810,Z 1258.607,A 0.000,B 0.000,C 90.000,E1 325.182} C_DIS
LIN {X 0.105,Y -506.538,Z 1258.603,A 0.000,B 0.000,C 90.000,E1 324.562} C_DIS
LIN {X -0.198,Y -504.244,Z 1258.598,A 0.000,B 0.000,C 90.000,E1 323.703} C_DIS
LIN {X 0.184,Y -502.836,Z 1258.593,A 0.000,B 0.000,C 90.000,E1 322.763} C_DIS
LIN {X -0.155,Y -502.276,Z 1258.588,A 0.000,B 0.000,C 90.000,E1 321.904} C_DIS
LIN {X -0.287,Y -502.617,Z 1258.568,A 0.000,B 0.000,C 90.000,E1 318.324} C_DIS
LIN {X 0.099,Y -502.984,Z 1258.560,A 0.000,B 0.000,C 90.000,E1 316.782} C_DIS
LIN {X -0.291,Y -503.517,Z 1258.547,A 0.000,B 0.000,C 90.000,E1 314.433} C_DIS
LIN {X -0.252,Y -503.839,Z 1258.538,A 0.000,B 0.000,C 90.000,E1 312.933} C_DIS
LIN {X 0.166,Y -504.172,Z 1258.530,A 0.000,B 0.000,C 90.000,E1 311.391} C_DIS
LIN {X -0.240,Y -504.466,Z 1258.520,A 0.000,B 0.000,C 90.000,E1 309.644} C_DIS
LIN {X -0.077,Y -505.047,Z 1258.507,A 0.000,B 0.000,C 90.000,E1 307.237} C_DIS
LIN {X -0.003,Y -505.361,Z 1258.497,A 0.000,B 0.000,C 90.000,E1 305.438} C_DIS
LIN {X 0.295,Y -505.497,Z 1258.489,A 0.000,B 0.000,C 90.000,E1 303.913} C_DIS
LIN {X 0.208,Y -505.521,Z 1258.479,A 0.000,B 0.000,C 90.000,E1 302.133} C_DIS
LIN {X -0.033,Y -505.414,Z 1258.470,A 0.000,B 0.000,C 90.000,E1 300.669} C_DIS
LIN {X 0.108,Y -505.285,Z 1258.459,A 0.000,B 0.000,C 90.000,E1 298.565} C_DIS
LIN {X 0.049,Y -505.248,Z 1258.455,A 0.000,B 0.000,C 90.000,E1 297.975} C_DIS
LIN {X 0.012,Y -504.920,Z 1258.442,A 0.000,B 0.000,C 90.000,E1 295.591} C_DIS
LIN {X 0.190,Y -504.905,Z 1258.434,A 0.000,B 0.000,C 90.000,E1 294.079} C_DIS
LIN {X -0.011,Y -504.794,Z 1258.429,A 0.000,B 0.000,C 90.000,E1 293.206} C_DIS
LIN {X 0.048,Y -504.254,Z 1258.419,A 0.000,B 0.000,C 90.000,E1 291.408} C_DIS
LIN {X 0.304,Y -503.911,Z 1258.414,A 0.000,B 0.000,C 90.000,E1 290.482} C_DIS
LIN {X 0.056,Y -502.623,Z 1258.402,A 0.000,B 0.000,C 90.000,E1 288.417} C_DIS
LIN {X 0.040,Y -501.820,Z 1258.396,A 0.000,B 0.000,C 90.000,E1 287.221} C_DIS
LIN {X 0.092,Y -501.086,Z 1258.391,A 0.000,B 0.000,C 90.000,E1 286.315} C_DIS
LIN {X -0.083,Y -499.936,Z 1258.384,A 0.000,B 0.000,C 90.000,E1 285.134} C_DIS
LIN {X -0.146,Y -498.552,Z 1258.377,A 0.000,B 0.000,C 90.000,E1 283.939} C_DIS
LIN {X 0.015,Y -496.905,Z 1258.371,A 0.000,B 0.000,C 90.000,E1 282.715} C_DIS
LIN {X -0.221,Y -494.991,Z 1258.364,A 0.000,B 0.000,C 90.000,E1 281.535} C_DIS
LIN {X 0.202,Y -487.984,Z 1258.335,A 0.000,B 0.000,C 90.000,E1 276.315} C_DIS
LIN {X -0.135,Y -485.809,Z 1258.282,A 0.000,B 0.000,C 90.000,E1 266.846} C_DIS
LIN {X -0.019,Y -486.065,Z 1258.274,A 0.000,B 0.000,C 90.000,E1 265.298} C_DIS
LIN {X 0.008,Y -486.074,Z 1258.269,A 0.000,B 0.000,C 90.000,E1 264.375} C_DIS
LIN {X -0.144,Y -485.921,Z 1258.262,A 0.000,B 0.000,C 90.000,E1 263.166} C_DIS
LIN {X 0.238,Y -485.546,Z 1258.255,A 0.000,B 0.000,C 90.000,E1 261.894} C_DIS
LIN {X -0.125,Y -484.354,Z 1258.245,A 0.000,B 0.000,C 90.000,E1 260.095} C_DIS
LIN {X -0.223,Y -482.620,Z 1258.231,A 0.000,B 0.000,C 90.000,E1 257.645} C_DIS
LIN {X -0.053,Y -481.989,Z 1258.226,A 0.000,B 0.000,C 90.000,E1 256.700} C_DIS
LIN {X 0.104,Y -480.587,Z 1258.212,A 0.000,B 0.000,C 90.000,E1 254.212} C_DIS
LIN {X 0.056,Y -479.512,Z 1258.202,A 0.000,B 0.000,C 90.000,E1 252.362} C_DIS
LIN {X 0.103,Y -478.352,Z 1258.190,A 0.000,B 0.000,C 90.000,E1 250.188} C_DIS
LIN {X 0.032,Y -477.564,Z 1258.181,A 0.000,B 0.000,C 90.000,E1 248.646} C_DIS
LIN {X -0.087,Y -476.388,Z 1258.169,A 0.000,B 0.000,C 90.000,E1 246.485} C_DIS
LIN {X 0.131,Y -474.956,Z 1258.157,A 0.000,B 0.000,C 90.000,E1 244.280} C_DIS
LIN {X 0.086,Y -473.479,Z 1258.145,A 0.000,B 0.000,C 90.000,E1 242.103} C_DIS
LIN {X -0.142,Y -472.207,Z 1258.135,A 0.000,B 0.000,C 90.000,E1 240.255} C_DIS
LIN {X -0.091,Y -471.267,Z 1258.128,A 0.000,B 0.000,C 90.000,E1 238.997} C_DIS
LIN {X 0.103,Y -469.992,Z 1258.119,A 0.000,B 0.000,C 90.000,E1 237.406} C_DIS
LIN {X -0.081,Y -468.247,Z 1258.107,A 0.000,B 0.000,C 90.000,E1 235.229} C_DIS
LIN {X 0.125,Y -466.630,Z 1258.093,A 0.000,B 0.000,C 90.000,E1 232.683} C_DIS
LIN {X -0.180,Y -465.401,Z 1258.079,A 0.000,B 0.000,C 90.000,E1 230.194} C_DIS
LIN {X -0.145,Y -464.723,Z 1258.070,A 0.000,B 0.000,C 90.000,E1 228.609} C_DIS
LIN {X 0.065,Y -464.322,Z 1258.065,A 0.000,B 0.000,C 90.000,E1 227.634} C_DIS
LIN {X 0.153,Y -463.172,Z 1258.052,A 0.000,B 0.000,C 90.000,E1 225.405} C_DIS
LIN {X 0.149,Y -461.791,Z 1258.031,A 0.000,B 0.000,C 90.000,E1 221.595} C_DIS
LIN {X 0.072,Y -462.847,Z 1258.006,A 0.000,B 0.000,C 90.000,E1 217.156} C_DIS
LIN {X -0.044,Y -466.202,Z 1257.980,A 0.000,B 0.000,C 90.000,E1 212.418} C_DIS
LIN {X -0.023,Y -469.988,Z 1257.961,A 0.000,B 0.000,C 90.000,E1 208.949} C_DIS
LIN {X -0.230,Y -471.575,Z 1257.954,A 0.000,B 0.000,C 90.000,E1 207.719} C_DIS
LIN {X -0.224,Y -475.508,Z 1257.937,A 0.000,B 0.000,C 90.000,E1 204.591} C_DIS
LIN {X -0.010,Y -479.277,Z 1257.923,A 0.000,B 0.000,C 90.000,E1 202.078} C_DIS
LIN {X 0.233,Y -484.696,Z 1257.906,A 0.000,B 0.000,C 90.000,E1 198.960} C_DIS
LIN {X -0.021,Y -488.394,Z 1257.895,A 0.000,B 0.000,C 90.000,E1 197.149} C_DIS
LIN {X 0.111,Y -491.554,Z 1257.887,A 0.000,B 0.000,C 90.000,E1 195.607} C_DIS
LIN {X 0.121,Y -496.009,Z 1257.875,A 0.000,B 0.000,C 90.000,E1 193.480} C_DIS
LIN {X 0.212,Y -499.995,Z 1257.865,A 0.000,B 0.000,C 90.000,E1 191.658} C_DIS
LIN {X -0.204,Y -504.086,Z 1257.855,A 0.000,B 0.000,C 90.000,E1 189.905} C_DIS
LIN {X -0.076,Y -507.513,Z 1257.847,A 0.000,B 0.000,C 90.000,E1 188.398} C_DIS
LIN {X 0.115,Y -511.049,Z 1257.838,A 0.000,B 0.000,C 90.000,E1 186.891} C_DIS
LIN {X 0.216,Y -515.127,Z 1257.828,A 0.000,B 0.000,C 90.000,E1 185.106} C_DIS
LIN {X -0.080,Y -518.516,Z 1257.820,A 0.000,B 0.000,C 90.000,E1 183.669} C_DIS
LIN {X 0.225,Y -521.191,Z 1257.814,A 0.000,B 0.000,C 90.000,E1 182.465} C_DIS
LIN {X 0.048,Y -523.793,Z 1257.807,A 0.000,B 0.000,C 90.000,E1 181.318} C_DIS
LIN {X -0.169,Y -527.598,Z 1257.798,A 0.000,B 0.000,C 90.000,E1 179.599} C_DIS
LIN {X 0.259,Y -530.092,Z 1257.791,A 0.000,B 0.000,C 90.000,E1 178.396} C_DIS
LIN {X 0.194,Y -533.045,Z 1257.783,A 0.000,B 0.000,C 90.000,E1 176.963} C_DIS
LIN {X 0.193,Y -534.703,Z 1257.779,A 0.000,B 0.000,C 90.000,E1 176.102} C_DIS
LIN {X 0.248,Y -536.730,Z 1257.772,A 0.000,B 0.000,C 90.000,E1 174.951} C_DIS
LIN {X -0.201,Y -539.159,Z 1257.764,A 0.000,B 0.000,C 90.000,E1 173.571} C_DIS
LIN {X 0.052,Y -541.700,Z 1257.755,A 0.000,B 0.000,C 90.000,E1 171.837} C_DIS
LIN {X 0.198,Y -542.895,Z 1257.750,A 0.000,B 0.000,C 90.000,E1 170.971} C_DIS
LIN {X 0.084,Y -544.685,Z 1257.742,A 0.000,B 0.000,C 90.000,E1 169.567} C_DIS
LIN {X -0.281,Y -545.657,Z 1257.737,A 0.000,B 0.000,C 90.000,E1 168.757} C_DIS
LIN {X 0.190,Y -547.048,Z 1257.730,A 0.000,B 0.000,C 90.000,E1 167.297} C_DIS
LIN {X -0.259,Y -548.324,Z 1257.722,A 0.000,B 0.000,C 90.000,E1 165.936} C_DIS
LIN {X 0.098,Y -549.962,Z 1257.712,A 0.000,B 0.000,C 90.000,E1 164.212} C_DIS
LIN {X 0.230,Y -552.479,Z 1257.702,A 0.000,B 0.000,C 90.000,E1 162.236} C_DIS
LIN {X 0.032,Y -555.200,Z 1257.694,A 0.000,B 0.000,C 90.000,E1 160.859} C_DIS
LIN {X 0.252,Y -559.020,Z 1257.686,A 0.000,B 0.000,C 90.000,E1 159.444} C_DIS
LIN {X -0.076,Y -561.879,Z 1257.681,A 0.000,B 0.000,C 90.000,E1 158.646} C_DIS
LIN {X 0.279,Y -567.509,Z 1257.674,A 0.000,B 0.000,C 90.000,E1 157.230} C_DIS
LIN {X -0.306,Y -574.289,Z 1257.666,A 0.000,B 0.000,C 90.000,E1 155.921} C_DIS
LIN {X -0.059,Y -589.035,Z 1257.652,A 0.000,B 0.000,C 90.000,E1 153.332} C_DIS
LIN {X -0.207,Y -595.316,Z 1257.646,A 0.000,B 0.000,C 90.000,E1 152.281} C_DIS
LIN {X 0.059,Y -599.937,Z 1257.641,A 0.000,B 0.000,C 90.000,E1 151.463} C_DIS
LIN {X 0.096,Y -605.128,Z 1257.636,A 0.000,B 0.000,C 90.000,E1 150.539} C_DIS
LIN {X -0.376,Y -611.516,Z 1257.630,A 0.000,B 0.000,C 90.000,E1 149.410} C_DIS
LIN {X 0.103,Y -617.030,Z 1257.624,A 0.000,B 0.000,C 90.000,E1 148.329} C_DIS
LIN {X -0.171,Y -620.965,Z 1257.620,A 0.000,B 0.000,C 90.000,E1 147.582} C_DIS
LIN {X 0.115,Y -624.811,Z 1257.616,A 0.000,B 0.000,C 90.000,E1 146.786} C_DIS
LIN {X -0.080,Y -626.676,Z 1257.613,A 0.000,B 0.000,C 90.000,E1 146.421} C_DIS
LIN {X 0.089,Y -632.498,Z 1257.606,A 0.000,B 0.000,C 90.000,E1 145.135} C_DIS
LIN {X 0.174,Y -636.610,Z 1257.601,A 0.000,B 0.000,C 90.000,E1 144.116} C_DIS
LIN {X 0.054,Y -638.594,Z 1257.598,A 0.000,B 0.000,C 90.000,E1 143.623} C_DIS
LIN {X 0.346,Y -641.282,Z 1257.594,A 0.000,B 0.000,C 90.000,E1 142.844} C_DIS
LIN {X -0.339,Y -644.679,Z 1257.588,A 0.000,B 0.000,C 90.000,E1 141.904} C_DIS
LIN {X -0.077,Y -647.752,Z 1257.583,A 0.000,B 0.000,C 90.000,E1 140.884} C_DIS
LIN {X 0.156,Y -651.311,Z 1257.576,A 0.000,B 0.000,C 90.000,E1 139.622} C_DIS
LIN {X -0.048,Y -654.729,Z 1257.569,A 0.000,B 0.000,C 90.000,E1 138.405} C_DIS
LIN {X 0.245,Y -658.017,Z 1257.562,A 0.000,B 0.000,C 90.000,E1 137.148} C_DIS
LIN {X 0.081,Y -663.121,Z 1257.551,A 0.000,B 0.000,C 90.000,E1 135.202} C_DIS
LIN {X 0.047,Y -667.228,Z 1257.543,A 0.000,B 0.000,C 90.000,E1 133.743} C_DIS
LIN {X 0.078,Y -671.368,Z 1257.535,A 0.000,B 0.000,C 90.000,E1 132.285} C_DIS
LIN {X 0.201,Y -674.760,Z 1257.528,A 0.000,B 0.000,C 90.000,E1 131.067} C_DIS
LIN {X -0.007,Y -679.359,Z 1257.519,A 0.000,B 0.000,C 90.000,E1 129.402} C_DIS
LIN {X -0.052,Y -683.064,Z 1257.511,A 0.000,B 0.000,C 90.000,E1 127.971} C_DIS
LIN {X -0.009,Y -686.794,Z 1257.503,A 0.000,B 0.000,C 90.000,E1 126.537} C_DIS
LIN {X -0.096,Y -689.680,Z 1257.496,A 0.000,B 0.000,C 90.000,E1 125.358} C_DIS
LIN {X -0.023,Y -691.786,Z 1257.491,A 0.000,B 0.000,C 90.000,E1 124.405} C_DIS
LIN {X 0.115,Y -694.256,Z 1257.485,A 0.000,B 0.000,C 90.000,E1 123.214} C_DIS
LIN {X -0.118,Y -696.169,Z 1257.479,A 0.000,B 0.000,C 90.000,E1 122.291} C_DIS
LIN {X -0.294,Y -698.432,Z 1257.473,A 0.000,B 0.000,C 90.000,E1 121.131} C_DIS
LIN {X -0.120,Y -699.645,Z 1257.469,A 0.000,B 0.000,C 90.000,E1 120.413} C_DIS
LIN {X 0.349,Y -701.507,Z 1257.462,A 0.000,B 0.000,C 90.000,E1 119.205} C_DIS
LIN {X 0.162,Y -703.039,Z 1257.456,A 0.000,B 0.000,C 90.000,E1 118.052} C_DIS
LIN {X -0.235,Y -703.807,Z 1257.452,A 0.000,B 0.000,C 90.000,E1 117.385} C_DIS
LIN {X 0.333,Y -704.212,Z 1257.449,A 0.000,B 0.000,C 90.000,E1 116.873} C_DIS
LIN {X -0.095,Y -704.566,Z 1257.444,A 0.000,B 0.000,C 90.000,E1 115.976} C_DIS
LIN {X 0.191,Y -704.612,Z 1257.443,A 0.000,B 0.000,C 90.000,E1 115.720} C_DIS
LIN {X -0.239,Y -704.169,Z 1257.438,A 0.000,B 0.000,C 90.000,E1 114.823} C_DIS
LIN {X -0.249,Y -703.956,Z 1257.437,A 0.000,B 0.000,C 90.000,E1 114.591} C_DIS
LIN {X 0.318,Y -703.097,Z 1257.434,A 0.000,B 0.000,C 90.000,E1 114.079} C_DIS
LIN {X -0.329,Y -702.355,Z 1257.433,A 0.000,B 0.000,C 90.000,E1 113.898} C_DIS
LIN {X 0.224,Y -700.475,Z 1257.430,A 0.000,B 0.000,C 90.000,E1 113.387} C_DIS
LIN {X 0.359,Y -699.717,Z 1257.429,A 0.000,B 0.000,C 90.000,E1 113.259} C_DIS
LIN {X -0.032,Y -695.505,Z 1257.427,A 0.000,B 0.000,C 90.000,E1 112.823} C_DIS
LIN {X 0.095,Y -694.148,Z 1257.426,A 0.000,B 0.000,C 90.000,E1 112.695} C_DIS
LIN {X 0.043,Y -692.108,Z 1257.426,A 0.000,B 0.000,C 90.000,E1 112.589} C_DIS
LIN {X 0.128,Y -687.484,Z 1257.425,A 0.000,B 0.000,C 90.000,E1 112.408} C_DIS
LIN {X -0.225,Y -682.480,Z 1257.424,A 0.000,B 0.000,C 90.000,E1 112.333} C_DIS
LIN {X -0.209,Y -677.960,Z 1257.424,A 0.000,B 0.000,C 90.000,E1 112.259} C_DIS
LIN {X 0.253,Y -674.613,Z 1257.424,A 0.000,B 0.000,C 90.000,E1 112.206} C_DIS
LIN {X 0.166,Y -671.046,Z 1257.423,A 0.000,B 0.000,C 90.000,E1 112.206} C_DIS
LIN {X 0.122,Y -630.357,Z 1257.423,A 0.000,B 0.000,C 90.000,E1 112.206} C_DIS
LIN {X -0.182,Y -628.168,Z 1257.423,A 0.000,B 0.000,C 90.000,E1 112.153} C_DIS
LIN {X -0.226,Y -628.085,Z 1257.423,A 0.000,B 0.000,C 90.000,E1 112.153} C_DIS
LIN {X 0.179,Y -626.529,Z 1257.422,A 0.000,B 0.000,C 90.000,E1 111.972} C_DIS
LIN {X 0.136,Y -626.509,Z 1257.422,A 0.000,B 0.000,C 90.000,E1 111.972} C_DIS
LIN {X 0.021,Y -626.446,Z 1257.422,A 0.000,B 0.000,C 90.000,E1 111.897} C_DIS
LIN {X 0.060,Y -626.818,Z 1257.421,A 0.000,B 0.000,C 90.000,E1 111.770} C_DIS
LIN {X 0.011,Y -628.687,Z 1257.419,A 0.000,B 0.000,C 90.000,E1 111.354} C_DIS
LIN {X -0.142,Y -636.705,Z 1257.411,A 0.000,B 0.000,C 90.000,E1 110.066} C_DIS
LIN {X -0.191,Y -641.417,Z 1257.407,A 0.000,B 0.000,C 90.000,E1 109.214} C_DIS
LIN {X 0.184,Y -646.273,Z 1257.401,A 0.000,B 0.000,C 90.000,E1 108.181} C_DIS
LIN {X -0.144,Y -652.186,Z 1257.394,A 0.000,B 0.000,C 90.000,E1 106.968} C_DIS
LIN {X 0.101,Y -655.458,Z 1257.390,A 0.000,B 0.000,C 90.000,E1 106.205} C_DIS
LIN {X 0.048,Y -657.490,Z 1257.387,A 0.000,B 0.000,C 90.000,E1 105.717} C_DIS
LIN {X -0.174,Y -659.245,Z 1257.385,A 0.000,B 0.000,C 90.000,E1 105.245} C_DIS
LIN {X 0.157,Y -661.470,Z 1257.381,A 0.000,B 0.000,C 90.000,E1 104.481} C_DIS
LIN {X -0.034,Y -662.696,Z 1257.378,A 0.000,B 0.000,C 90.000,E1 104.008} C_DIS
LIN {X -0.306,Y -664.028,Z 1257.374,A 0.000,B 0.000,C 90.000,E1 103.300} C_DIS
LIN {X 0.167,Y -664.592,Z 1257.371,A 0.000,B 0.000,C 90.000,E1 102.771} C_DIS
LIN {X -0.006,Y -664.893,Z 1257.368,A 0.000,B 0.000,C 90.000,E1 102.299} C_DIS
LIN {X -0.178,Y -664.936,Z 1257.366,A 0.000,B 0.000,C 90.000,E1 101.827} C_DIS
LIN {X 0.299,Y -664.683,Z 1257.363,A 0.000,B 0.000,C 90.000,E1 101.299} C_DIS
LIN {X -0.006,Y -664.214,Z 1257.360,A 0.000,B 0.000,C 90.000,E1 100.838} C_DIS
LIN {X -0.096,Y -663.945,Z 1257.359,A 0.000,B 0.000,C 90.000,E1 100.602} C_DIS
LIN {X 0.254,Y -663.017,Z 1257.356,A 0.000,B 0.000,C 90.000,E1 100.084} C_DIS
LIN {X -0.038,Y -661.204,Z 1257.352,A 0.000,B 0.000,C 90.000,E1 99.378} C_DIS
LIN {X 0.299,Y -659.600,Z 1257.349,A 0.000,B 0.000,C 90.000,E1 98.859} C_DIS
LIN {X -0.022,Y -657.511,Z 1257.347,A 0.000,B 0.000,C 90.000,E1 98.398} C_DIS
LIN {X 0.279,Y -654.489,Z 1257.343,A 0.000,B 0.000,C 90.000,E1 97.757} C_DIS
LIN {X -0.185,Y -650.944,Z 1257.340,A 0.000,B 0.000,C 90.000,E1 97.182} C_DIS
LIN {X 0.087,Y -647.708,Z 1257.337,A 0.000,B 0.000,C 90.000,E1 96.663} C_DIS
LIN {X -0.305,Y -644.081,Z 1257.334,A 0.000,B 0.000,C 90.000,E1 96.201} C_DIS
LIN {X -0.205,Y -639.058,Z 1257.331,A 0.000,B 0.000,C 90.000,E1 95.568} C_DIS
LIN {X -0.016,Y -634.522,Z 1257.328,A 0.000,B 0.000,C 90.000,E1 95.049} C_DIS
LIN {X 0.220,Y -629.595,Z 1257.325,A 0.000,B 0.000,C 90.000,E1 94.531} C_DIS
LIN {X -0.085,Y -623.092,Z 1257.322,A 0.000,B 0.000,C 90.000,E1 93.955} C_DIS
LIN {X -0.202,Y -616.221,Z 1257.319,A 0.000,B 0.000,C 90.000,E1 93.383} C_DIS
LIN {X 0.078,Y -608.910,Z 1257.316,A 0.000,B 0.000,C 90.000,E1 92.808} C_DIS
LIN {X 0.032,Y -601.293,Z 1257.313,A 0.000,B 0.000,C 90.000,E1 92.293} C_DIS
LIN {X 0.042,Y -595.048,Z 1257.311,A 0.000,B 0.000,C 90.000,E1 91.892} C_DIS
LIN {X 0.103,Y -590.126,Z 1257.309,A 0.000,B 0.000,C 90.000,E1 91.604} C_DIS
LIN {X 0.185,Y -583.240,Z 1257.307,A 0.000,B 0.000,C 90.000,E1 91.260} C_DIS
LIN {X -0.031,Y -571.267,Z 1257.304,A 0.000,B 0.000,C 90.000,E1 90.802} C_DIS
LIN {X 0.229,Y -569.295,Z 1257.304,A 0.000,B 0.000,C 90.000,E1 90.630} C_DIS
LIN {X 0.131,Y -568.001,Z 1257.303,A 0.000,B 0.000,C 90.000,E1 90.516} C_DIS
LIN {X -0.280,Y -567.837,Z 1257.303,A 0.000,B 0.000,C 90.000,E1 90.516} C_DIS
LIN {X -0.016,Y -567.400,Z 1257.299,A 0.000,B 0.000,C 90.000,E1 89.885} C_DIS
LIN {X 0.028,Y -568.012,Z 1257.293,A 0.000,B 0.000,C 90.000,E1 88.797} C_DIS
LIN {X 0.211,Y -569.353,Z 1257.284,A 0.000,B 0.000,C 90.000,E1 87.135} C_DIS
LIN {X -0.267,Y -571.635,Z 1257.271,A 0.000,B 0.000,C 90.000,E1 84.723} C_DIS
LIN {X 0.264,Y -573.652,Z 1257.260,A 0.000,B 0.000,C 90.000,E1 82.761} C_DIS
LIN {X -0.047,Y -575.139,Z 1257.252,A 0.000,B 0.000,C 90.000,E1 81.432} C_DIS
LIN {X -0.247,Y -576.511,Z 1257.245,A 0.000,B 0.000,C 90.000,E1 80.095} C_DIS
LIN {X -0.072,Y -577.386,Z 1257.239,A 0.000,B 0.000,C 90.000,E1 78.993} C_DIS
LIN {X 0.090,Y -578.676,Z 1257.230,A 0.000,B 0.000,C 90.000,E1 77.353} C_DIS
LIN {X 0.071,Y -579.957,Z 1257.219,A 0.000,B 0.000,C 90.000,E1 75.463} C_DIS
LIN {X 0.197,Y -580.795,Z 1257.212,A 0.000,B 0.000,C 90.000,E1 74.102} C_DIS
LIN {X -0.010,Y -581.868,Z 1257.201,A 0.000,B 0.000,C 90.000,E1 72.236} C_DIS
LIN {X 0.099,Y -582.586,Z 1257.195,A 0.000,B 0.000,C 90.000,E1 71.148} C_DIS
LIN {X -0.131,Y -583.359,Z 1257.188,A 0.000,B 0.000,C 90.000,E1 69.826} C_DIS
LIN {X -0.023,Y -584.659,Z 1257.176,A 0.000,B 0.000,C 90.000,E1 67.667} C_DIS
LIN {X -0.182,Y -586.351,Z 1257.164,A 0.000,B 0.000,C 90.000,E1 65.537} C_DIS
LIN {X 0.180,Y -587.647,Z 1257.155,A 0.000,B 0.000,C 90.000,E1 63.896} C_DIS
LIN {X 0.302,Y -589.075,Z 1257.146,A 0.000,B 0.000,C 90.000,E1 62.281} C_DIS
LIN {X 0.042,Y -590.466,Z 1257.139,A 0.000,B 0.000,C 90.000,E1 60.973} C_DIS
LIN {X -0.304,Y -592.107,Z 1257.130,A 0.000,B 0.000,C 90.000,E1 59.410} C_DIS
LIN {X -0.118,Y -593.213,Z 1257.124,A 0.000,B 0.000,C 90.000,E1 58.329} C_DIS
LIN {X -0.024,Y -594.518,Z 1257.117,A 0.000,B 0.000,C 90.000,E1 56.993} C_DIS
LIN {X 0.025,Y -596.334,Z 1257.106,A 0.000,B 0.000,C 90.000,E1 55.135} C_DIS
LIN {X 0.090,Y -597.691,Z 1257.098,A 0.000,B 0.000,C 90.000,E1 53.543} C_DIS
LIN {X 0.072,Y -599.196,Z 1257.087,A 0.000,B 0.000,C 90.000,E1 51.698} C_DIS
LIN {X 0.338,Y -600.117,Z 1257.080,A 0.000,B 0.000,C 90.000,E1 50.356} C_DIS
LIN {X -0.010,Y -600.568,Z 1257.074,A 0.000,B 0.000,C 90.000,E1 49.337} C_DIS
LIN {X -0.018,Y -601.102,Z 1257.068,A 0.000,B 0.000,C 90.000,E1 48.286} C_DIS
LIN {X -0.170,Y -601.499,Z 1257.061,A 0.000,B 0.000,C 90.000,E1 46.986} C_DIS
LIN {X 0.088,Y -601.901,Z 1257.054,A 0.000,B 0.000,C 90.000,E1 45.648} C_DIS
LIN {X -0.081,Y -601.835,Z 1257.046,A 0.000,B 0.000,C 90.000,E1 44.352} C_DIS
LIN {X -0.053,Y -601.631,Z 1257.041,A 0.000,B 0.000,C 90.000,E1 43.299} C_DIS
LIN {X -0.206,Y -601.160,Z 1257.033,A 0.000,B 0.000,C 90.000,E1 42.000} C_DIS
LIN {X 0.030,Y -600.673,Z 1257.026,A 0.000,B 0.000,C 90.000,E1 40.663} C_DIS
LIN {X -0.292,Y -599.723,Z 1257.017,A 0.000,B 0.000,C 90.000,E1 39.116} C_DIS
LIN {X 0.202,Y -598.952,Z 1257.011,A 0.000,B 0.000,C 90.000,E1 38.016} C_DIS
LIN {X 0.082,Y -598.260,Z 1257.007,A 0.000,B 0.000,C 90.000,E1 37.237} C_DIS
LIN {X -0.055,Y -596.616,Z 1257.000,A 0.000,B 0.000,C 90.000,E1 35.931} C_DIS
LIN {X -0.313,Y -595.072,Z 1256.994,A 0.000,B 0.000,C 90.000,E1 34.898} C_DIS
LIN {X 0.134,Y -594.169,Z 1256.991,A 0.000,B 0.000,C 90.000,E1 34.326} C_DIS
LIN {X -0.156,Y -592.116,Z 1256.985,A 0.000,B 0.000,C 90.000,E1 33.293} C_DIS
LIN {X 0.140,Y -590.224,Z 1256.980,A 0.000,B 0.000,C 90.000,E1 32.467} C_DIS
LIN {X -0.018,Y -587.251,Z 1256.975,A 0.000,B 0.000,C 90.000,E1 31.416} C_DIS
LIN {X 0.220,Y -584.627,Z 1256.970,A 0.000,B 0.000,C 90.000,E1 30.590} C_DIS
LIN {X -0.033,Y -582.616,Z 1256.967,A 0.000,B 0.000,C 90.000,E1 30.079} C_DIS
LIN {X -0.008,Y -580.414,Z 1256.964,A 0.000,B 0.000,C 90.000,E1 29.539} C_DIS
LIN {X -0.143,Y -576.724,Z 1256.960,A 0.000,B 0.000,C 90.000,E1 28.743} C_DIS
LIN {X 0.257,Y -573.384,Z 1256.956,A 0.000,B 0.000,C 90.000,E1 28.025} C_DIS
LIN {X 0.018,Y -571.256,Z 1256.954,A 0.000,B 0.000,C 90.000,E1 27.641} C_DIS
LIN {X 0.105,Y -567.341,Z 1256.950,A 0.000,B 0.000,C 90.000,E1 26.950} C_DIS
LIN {X 0.001,Y -563.949,Z 1256.947,A 0.000,B 0.000,C 90.000,E1 26.411} C_DIS
LIN {X -0.073,Y -558.505,Z 1256.942,A 0.000,B 0.000,C 90.000,E1 25.591} C_DIS
LIN {X -0.090,Y -553.527,Z 1256.938,A 0.000,B 0.000,C 90.000,E1 24.899} C_DIS
LIN {X -0.035,Y -549.231,Z 1256.935,A 0.000,B 0.000,C 90.000,E1 24.335} C_DIS
LIN {X -0.010,Y -544.690,Z 1256.932,A 0.000,B 0.000,C 90.000,E1 23.770} C_DIS
LIN {X -0.019,Y -539.870,Z 1256.929,A 0.000,B 0.000,C 90.000,E1 23.206} C_DIS
LIN {X 0.082,Y -530.954,Z 1256.923,A 0.000,B 0.000,C 90.000,E1 22.206} C_DIS
LIN {X -0.215,Y -524.311,Z 1256.920,A 0.000,B 0.000,C 90.000,E1 21.535} C_DIS
LIN {X 0.228,Y -516.408,Z 1256.915,A 0.000,B 0.000,C 90.000,E1 20.663} C_DIS
LIN {X -0.123,Y -507.131,Z 1256.910,A 0.000,B 0.000,C 90.000,E1 19.758} C_DIS
LIN {X 0.166,Y -496.158,Z 1256.904,A 0.000,B 0.000,C 90.000,E1 18.671} C_DIS
LIN {X -0.070,Y -484.571,Z 1256.898,A 0.000,B 0.000,C 90.000,E1 17.638} C_DIS
LIN {X -0.145,Y -477.229,Z 1256.894,A 0.000,B 0.000,C 90.000,E1 16.985} C_DIS
LIN {X -0.075,Y -462.384,Z 1256.887,A 0.000,B 0.000,C 90.000,E1 15.662} C_DIS
LIN {X -0.225,Y -444.680,Z 1256.878,A 0.000,B 0.000,C 90.000,E1 14.064} C_DIS
LIN {X 0.006,Y -428.851,Z 1256.869,A 0.000,B 0.000,C 90.000,E1 12.479} C_DIS
LIN {X 0.103,Y -414.477,Z 1256.861,A 0.000,B 0.000,C 90.000,E1 10.950} C_DIS
LIN {X -0.132,Y -401.688,Z 1256.853,A 0.000,B 0.000,C 90.000,E1 9.557} C_DIS
LIN {X -0.109,Y -397.933,Z 1256.850,A 0.000,B 0.000,C 90.000,E1 9.095} C_DIS
LIN {X -0.042,Y -396.740,Z 1256.850,A 0.000,B 0.000,C 90.000,E1 8.916} C_DIS
LIN {X -0.136,Y -394.635,Z 1256.848,A 0.000,B 0.000,C 90.000,E1 8.568} C_DIS
LIN {X -0.174,Y -394.606,Z 1256.848,A 0.000,B 0.000,C 90.000,E1 8.568} C_DIS
LIN {X 0.190,Y -394.500,Z 1256.847,A 0.000,B 0.000,C 90.000,E1 8.454} C_DIS
LIN {X 0.152,Y -394.509,Z 1256.847,A 0.000,B 0.000,C 90.000,E1 8.454} C_DIS
LIN {X -0.071,Y -396.106,Z 1256.845,A 0.000,B 0.000,C 90.000,E1 8.106} C_DIS
LIN {X 0.103,Y -396.770,Z 1256.844,A 0.000,B 0.000,C 90.000,E1 7.992} C_DIS
LIN {X -0.126,Y -400.931,Z 1256.842,A 0.000,B 0.000,C 90.000,E1 7.644} C_DIS
LIN {X 0.179,Y -406.719,Z 1256.840,A 0.000,B 0.000,C 90.000,E1 7.182} C_DIS
LIN {X 0.179,Y -412.892,Z 1256.838,A 0.000,B 0.000,C 90.000,E1 6.777} C_DIS
LIN {X -0.143,Y -419.440,Z 1256.835,A 0.000,B 0.000,C 90.000,E1 6.372} C_DIS
LIN {X 0.189,Y -427.490,Z 1256.832,A 0.000,B 0.000,C 90.000,E1 5.739} C_DIS
LIN {X 0.005,Y -435.413,Z 1256.829,A 0.000,B 0.000,C 90.000,E1 5.163} C_DIS
LIN {X 0.049,Y -445.992,Z 1256.824,A 0.000,B 0.000,C 90.000,E1 4.302} C_DIS
LIN {X -0.035,Y -455.261,Z 1256.820,A 0.000,B 0.000,C 90.000,E1 3.555} C_DIS
LIN {X 0.050,Y -461.273,Z 1256.817,A 0.000,B 0.000,C 90.000,E1 3.037} C_DIS
LIN {X -0.068,Y -468.492,Z 1256.813,A 0.000,B 0.000,C 90.000,E1 2.407} C_DIS
LIN {X -0.130,Y -472.846,Z 1256.811,A 0.000,B 0.000,C 90.000,E1 2.007} C_DIS
LIN {X -0.063,Y -479.531,Z 1256.807,A 0.000,B 0.000,C 90.000,E1 1.318} C_DIS
LIN {X -0.210,Y -485.977,Z 1256.803,A 0.000,B 0.000,C 90.000,E1 0.630} C_DIS
LIN {X 0.000,Y -491.050,Z 1256.800,A 0.000,B 0.000,C 90.000,E1 360.000} C_DIS
LIN {X 0.032,Y -495.217,Z 1256.797,A 0.000,B 0.000,C 90.000,E1 359.484} C_DIS
LIN {X -0.067,Y -500.725,Z 1256.793,A 0.000,B 0.000,C 90.000,E1 358.740} C_DIS
LIN {X 0.097,Y -506.822,Z 1256.788,A 0.000,B 0.000,C 90.000,E1 357.822} C_DIS
LIN {X -0.108,Y -510.692,Z 1256.785,A 0.000,B 0.000,C 90.000,E1 357.249} C_DIS
LIN {X 0.173,Y -516.051,Z 1256.780,A 0.000,B 0.000,C 90.000,E1 356.331} C_DIS
LIN {X 0.064,Y -519.357,Z 1256.776,A 0.000,B 0.000,C 90.000,E1 355.755} C_DIS
LIN {X 0.212,Y -523.193,Z 1256.772,A 0.000,B 0.000,C 90.000,E1 355.008} C_DIS
LIN {X 0.158,Y -526.062,Z 1256.769,A 0.000,B 0.000,C 90.000,E1 354.432} C_DIS
LIN {X -0.158,Y -529.391,Z 1256.765,A 0.000,B 0.000,C 90.000,E1 353.742} C_DIS
LIN {X 0.110,Y -531.300,Z 1256.763,A 0.000,B 0.000,C 90.000,E1 353.280} C_DIS
LIN {X 0.151,Y -534.710,Z 1256.758,A 0.000,B 0.000,C 90.000,E1 352.413} C_DIS
LIN {X 0.225,Y -537.821,Z 1256.753,A 0.000,B 0.000,C 90.000,E1 351.546} C_DIS
LIN {X -0.203,Y -540.756,Z 1256.748,A 0.000,B 0.000,C 90.000,E1 350.735} C_DIS
LIN {X 0.023,Y -543.298,Z 1256.744,A 0.000,B 0.000,C 90.000,E1 349.859} C_DIS
LIN {X -0.266,Y -546.462,Z 1256.737,A 0.000,B 0.000,C 90.000,E1 348.757} C_DIS
LIN {X 0.125,Y -549.206,Z 1256.731,A 0.000,B 0.000,C 90.000,E1 347.589} C_DIS
LIN {X 0.256,Y -552.313,Z 1256.723,A 0.000,B 0.000,C 90.000,E1 346.172} C_DIS
LIN {X 0.065,Y -553.899,Z 1256.719,A 0.000,B 0.000,C 90.000,E1 345.353} C_DIS
LIN {X 0.300,Y -555.771,Z 1256.713,A 0.000,B 0.000,C 90.000,E1 344.212} C_DIS
LIN {X -0.119,Y -557.416,Z 1256.706,A 0.000,B 0.000,C 90.000,E1 343.142} C_DIS
LIN {X -0.118,Y -558.460,Z 1256.702,A 0.000,B 0.000,C 90.000,E1 342.308} C_DIS
LIN {X 0.187,Y -559.512,Z 1256.696,A 0.000,B 0.000,C 90.000,E1 341.167} C_DIS
LIN {X 0.160,Y -560.082,Z 1256.689,A 0.000,B 0.000,C 90.000,E1 340.061} C_DIS
LIN {X -0.159,Y -560.223,Z 1256.685,A 0.000,B 0.000,C 90.000,E1 339.263} C_DIS
LIN {X 0.044,Y -559.980,Z 1256.680,A 0.000,B 0.000,C 90.000,E1 338.411} C_DIS
LIN {X 0.143,Y -559.686,Z 1256.677,A 0.000,B 0.000,C 90.000,E1 337.847} C_DIS
LIN {X -0.184,Y -558.921,Z 1256.672,A 0.000,B 0.000,C 90.000,E1 337.050} C_DIS
LIN {X 0.210,Y -557.864,Z 1256.668,A 0.000,B 0.000,C 90.000,E1 336.177} C_DIS
LIN {X 0.083,Y -556.579,Z 1256.663,A 0.000,B 0.000,C 90.000,E1 335.357} C_DIS
LIN {X 0.006,Y -553.734,Z 1256.656,A 0.000,B 0.000,C 90.000,E1 333.973} C_DIS
LIN {X -0.149,Y -550.686,Z 1256.649,A 0.000,B 0.000,C 90.000,E1 332.871} C_DIS
LIN {X -0.102,Y -547.886,Z 1256.645,A 0.000,B 0.000,C 90.000,E1 332.025} C_DIS
LIN {X 0.160,Y -545.764,Z 1256.641,A 0.000,B 0.000,C 90.000,E1 331.435} C_DIS
LIN {X 0.153,Y -542.048,Z 1256.637,A 0.000,B 0.000,C 90.000,E1 330.589} C_DIS
LIN {X 0.095,Y -537.632,Z 1256.632,A 0.000,B 0.000,C 90.000,E1 329.744} C_DIS
LIN {X -0.189,Y -534.350,Z 1256.629,A 0.000,B 0.000,C 90.000,E1 329.203} C_DIS
LIN {X 0.203,Y -525.982,Z 1256.622,A 0.000,B 0.000,C 90.000,E1 327.867} C_DIS
LIN {X -0.059,Y -515.464,Z 1256.613,A 0.000,B 0.000,C 90.000,E1 326.294} C_DIS
LIN {X 0.222,Y -512.100,Z 1256.609,A 0.000,B 0.000,C 90.000,E1 325.674} C_DIS
LIN {X -0.189,Y -509.387,Z 1256.606,A 0.000,B 0.000,C 90.000,E1 325.182} C_DIS
LIN {X 0.045,Y -506.992,Z 1256.603,A 0.000,B 0.000,C 90.000,E1 324.562} C_DIS
LIN {X -0.253,Y -504.600,Z 1256.598,A 0.000,B 0.000,C 90.000,E1 323.703} C_DIS
LIN {X 0.134,Y -503.172,Z 1256.593,A 0.000,B 0.000,C 90.000,E1 322.763} C_DIS
LIN {X -0.202,Y -502.610,Z 1256.588,A 0.000,B 0.000,C 90.000,E1 321.904} C_DIS
LIN {X 0.017,Y -503.016,Z 1256.568,A 0.000,B 0.000,C 90.000,E1 318.286} C_DIS
LIN {X -0.071,Y -503.484,Z 1256.558,A 0.000,B 0.000,C 90.000,E1 316.500} C_DIS
LIN {X 0.190,Y -503.882,Z 1256.548,A 0.000,B 0.000,C 90.000,E1 314.676} C_DIS
LIN {X -0.129,Y -504.212,Z 1256.540,A 0.000,B 0.000,C 90.000,E1 313.218} C_DIS
LIN {X 0.172,Y -504.655,Z 1256.530,A 0.000,B 0.000,C 90.000,E1 311.391} C_DIS
LIN {X -0.222,Y -504.964,Z 1256.520,A 0.000,B 0.000,C 90.000,E1 309.644} C_DIS
LIN {X 0.060,Y -505.441,Z 1256.509,A 0.000,B 0.000,C 90.000,E1 307.523} C_DIS
LIN {X 0.249,Y -505.798,Z 1256.500,A 0.000,B 0.000,C 90.000,E1 306.011} C_DIS
LIN {X 0.142,Y -506.005,Z 1256.492,A 0.000,B 0.000,C 90.000,E1 304.532} C_DIS
LIN {X -0.142,Y -506.039,Z 1256.485,A 0.000,B 0.000,C 90.000,E1 303.372} C_DIS
LIN {X -0.105,Y -506.055,Z 1256.477,A 0.000,B 0.000,C 90.000,E1 301.878} C_DIS
LIN {X 0.043,Y -505.989,Z 1256.470,A 0.000,B 0.000,C 90.000,E1 300.669} C_DIS
LIN {X 0.127,Y -505.904,Z 1256.461,A 0.000,B 0.000,C 90.000,E1 298.871} C_DIS
LIN {X 0.146,Y -505.834,Z 1256.456,A 0.000,B 0.000,C 90.000,E1 297.975} C_DIS
LIN {X 0.043,Y -505.541,Z 1256.444,A 0.000,B 0.000,C 90.000,E1 295.899} C_DIS
LIN {X 0.227,Y -505.528,Z 1256.436,A 0.000,B 0.000,C 90.000,E1 294.387} C_DIS
LIN {X 0.121,Y -505.463,Z 1256.429,A 0.000,B 0.000,C 90.000,E1 293.206} C_DIS
LIN {X 0.106,Y -505.077,Z 1256.421,A 0.000,B 0.000,C 90.000,E1 291.716} C_DIS
LIN {X -0.103,Y -504.414,Z 1256.412,A 0.000,B 0.000,C 90.000,E1 290.248} C_DIS
LIN {X 0.228,Y -503.335,Z 1256.399,A 0.000,B 0.000,C 90.000,E1 287.819} C_DIS
LIN {X 0.225,Y -502.768,Z 1256.393,A 0.000,B 0.000,C 90.000,E1 286.622} C_DIS
LIN {X 0.140,Y -501.799,Z 1256.384,A 0.000,B 0.000,C 90.000,E1 285.134} C_DIS
LIN {X 0.106,Y -500.862,Z 1256.378,A 0.000,B 0.000,C 90.000,E1 283.939} C_DIS
LIN {X -0.258,Y -499.470,Z 1256.369,A 0.000,B 0.000,C 90.000,E1 282.479} C_DIS
LIN {X -0.130,Y -497.620,Z 1256.359,A 0.000,B 0.000,C 90.000,E1 280.658} C_DIS
LIN {X -0.233,Y -495.910,Z 1256.349,A 0.000,B 0.000,C 90.000,E1 278.859} C_DIS
LIN {X -0.046,Y -494.099,Z 1256.337,A 0.000,B 0.000,C 90.000,E1 276.720} C_DIS
LIN {X -0.124,Y -492.490,Z 1256.324,A 0.000,B 0.000,C 90.000,E1 274.302} C_DIS
LIN {X -0.160,Y -491.312,Z 1256.312,A 0.000,B 0.000,C 90.000,E1 272.178} C_DIS
LIN {X 0.242,Y -490.228,Z 1256.300,A 0.000,B 0.000,C 90.000,E1 270.000} C_DIS
LIN {X 0.102,Y -489.710,Z 1256.293,A 0.000,B 0.000,C 90.000,E1 268.797} C_DIS
LIN {X -0.010,Y -488.970,Z 1256.282,A 0.000,B 0.000,C 90.000,E1 266.674} C_DIS
LIN {X 0.030,Y -488.415,Z 1256.271,A 0.000,B 0.000,C 90.000,E1 264.837} C_DIS
LIN {X -0.216,Y -487.775,Z 1256.263,A 0.000,B 0.000,C 90.000,E1 263.337} C_DIS
LIN {X 0.200,Y -487.076,Z 1256.256,A 0.000,B 0.000,C 90.000,E1 262.064} C_DIS
LIN {X 0.121,Y -486.006,Z 1256.249,A 0.000,B 0.000,C 90.000,E1 260.849} C_DIS
LIN {X -0.108,Y -484.609,Z 1256.241,A 0.000,B 0.000,C 90.000,E1 259.342} C_DIS
LIN {X -0.243,Y -482.591,Z 1256.225,A 0.000,B 0.000,C 90.000,E1 256.589} C_DIS
LIN {X 0.069,Y -481.325,Z 1256.213,A 0.000,B 0.000,C 90.000,E1 254.393} C_DIS
LIN {X 0.025,Y -480.122,Z 1256.201,A 0.000,B 0.000,C 90.000,E1 252.236} C_DIS
LIN {X 0.093,Y -478.958,Z 1256.189,A 0.000,B 0.000,C 90.000,E1 250.061} C_DIS
LIN {X -0.124,Y -478.328,Z 1256.182,A 0.000,B 0.000,C 90.000,E1 248.847} C_DIS
LIN {X -0.047,Y -477.181,Z 1256.170,A 0.000,B 0.000,C 90.000,E1 246.666} C_DIS
LIN {X 0.070,Y -476.322,Z 1256.163,A 0.000,B 0.000,C 90.000,E1 245.409} C_DIS
LIN {X 0.140,Y -475.325,Z 1256.155,A 0.000,B 0.000,C 90.000,E1 243.845} C_DIS
LIN {X 0.140,Y -474.034,Z 1256.144,A 0.000,B 0.000,C 90.000,E1 241.975} C_DIS
LIN {X -0.076,Y -472.719,Z 1256.134,A 0.000,B 0.000,C 90.000,E1 240.127} C_DIS
LIN {X -0.194,Y -471.999,Z 1256.129,A 0.000,B 0.000,C 90.000,E1 239.203} C_DIS
LIN {X 0.267,Y -470.708,Z 1256.120,A 0.000,B 0.000,C 90.000,E1 237.582} C_DIS
LIN {X 0.003,Y -468.665,Z 1256.106,A 0.000,B 0.000,C 90.000,E1 235.102} C_DIS
LIN {X -0.258,Y -466.700,Z 1256.089,A 0.000,B 0.000,C 90.000,E1 231.984} C_DIS
LIN {X -0.032,Y -465.652,Z 1256.076,A 0.000,B 0.000,C 90.000,E1 229.747} C_DIS
LIN {X -0.055,Y -465.046,Z 1256.069,A 0.000,B 0.000,C 90.000,E1 228.485} C_DIS
LIN {X -0.189,Y -464.578,Z 1256.064,A 0.000,B 0.000,C 90.000,E1 227.553} C_DIS
LIN {X -0.268,Y -463.839,Z 1256.057,A 0.000,B 0.000,C 90.000,E1 226.296} C_DIS
LIN {X 0.133,Y -462.705,Z 1256.045,A 0.000,B 0.000,C 90.000,E1 224.028} C_DIS
LIN {X -0.124,Y -462.084,Z 1256.022,A 0.000,B 0.000,C 90.000,E1 219.930} C_DIS
LIN {X -0.036,Y -463.241,Z 1256.004,A 0.000,B 0.000,C 90.000,E1 216.744} C_DIS
LIN {X 0.122,Y -466.438,Z 1255.979,A 0.000,B 0.000,C 90.000,E1 212.291} C_DIS
LIN {X -0.001,Y -469.835,Z 1255.962,A 0.000,B 0.000,C 90.000,E1 209.155} C_DIS
LIN {X 0.013,Y -471.439,Z 1255.955,A 0.000,B 0.000,C 90.000,E1 207.897} C_DIS
LIN {X 0.005,Y -475.344,Z 1255.938,A 0.000,B 0.000,C 90.000,E1 204.771} C_DIS
LIN {X 0.028,Y -479.070,Z 1255.924,A 0.000,B 0.000,C 90.000,E1 202.280} C_DIS
LIN {X -0.169,Y -485.009,Z 1255.905,A 0.000,B 0.000,C 90.000,E1 198.906} C_DIS
LIN {X 0.038,Y -488.143,Z 1255.896,A 0.000,B 0.000,C 90.000,E1 197.347} C_DIS
LIN {X -0.160,Y -491.339,Z 1255.888,A 0.000,B 0.000,C 90.000,E1 195.843} C_DIS
LIN {X -0.043,Y -495.843,Z 1255.876,A 0.000,B 0.000,C 90.000,E1 193.703} C_DIS
LIN {X 0.030,Y -499.858,Z 1255.866,A 0.000,B 0.000,C 90.000,E1 191.883} C_DIS
LIN {X -0.057,Y -504.696,Z 1255.854,A 0.000,B 0.000,C 90.000,E1 189.792} C_DIS
LIN {X 0.162,Y -508.146,Z 1255.846,A 0.000,B 0.000,C 90.000,E1 188.276} C_DIS
LIN {X -0.211,Y -511.738,Z 1255.838,A 0.000,B 0.000,C 90.000,E1 186.834} C_DIS
LIN {X -0.012,Y -515.219,Z 1255.830,A 0.000,B 0.000,C 90.000,E1 185.334} C_DIS
LIN {X 0.207,Y -518.679,Z 1255.822,A 0.000,B 0.000,C 90.000,E1 183.841} C_DIS
LIN {X -0.007,Y -521.431,Z 1255.815,A 0.000,B 0.000,C 90.000,E1 182.694} C_DIS
LIN {X 0.224,Y -526.029,Z 1255.804,A 0.000,B 0.000,C 90.000,E1 180.630} C_DIS
LIN {X 0.080,Y -529.280,Z 1255.796,A 0.000,B 0.000,C 90.000,E1 179.198} C_DIS
LIN {X 0.019,Y -531.143,Z 1255.791,A 0.000,B 0.000,C 90.000,E1 178.339} C_DIS
LIN {X -0.018,Y -533.569,Z 1255.784,A 0.000,B 0.000,C 90.000,E1 177.192} C_DIS
LIN {X 0.014,Y -536.373,Z 1255.776,A 0.000,B 0.000,C 90.000,E1 175.755} C_DIS
LIN {X 0.050,Y -538.415,Z 1255.770,A 0.000,B 0.000,C 90.000,E1 174.609} C_DIS
LIN {X 0.158,Y -540.433,Z 1255.764,A 0.000,B 0.000,C 90.000,E1 173.457} C_DIS
LIN {X -0.022,Y -543.511,Z 1255.753,A 0.000,B 0.000,C 90.000,E1 171.489} C_DIS
LIN {X -0.217,Y -545.426,Z 1255.745,A 0.000,B 0.000,C 90.000,E1 170.095} C_DIS
LIN {X 0.160,Y -546.873,Z 1255.739,A 0.000,B 0.000,C 90.000,E1 168.926} C_DIS
LIN {X 0.027,Y -548.121,Z 1255.732,A 0.000,B 0.000,C 90.000,E1 167.813} C_DIS
LIN {X 0.013,Y -549.602,Z 1255.725,A 0.000,B 0.000,C 90.000,E1 166.408} C_DIS
LIN {X 0.086,Y -552.067,Z 1255.712,A 0.000,B 0.000,C 90.000,E1 164.157} C_DIS
LIN {X -0.010,Y -554.398,Z 1255.703,A 0.000,B 0.000,C 90.000,E1 162.489} C_DIS
LIN {X -0.002,Y -557.118,Z 1255.695,A 0.000,B 0.000,C 90.000,E1 161.094} C_DIS
LIN {X 0.062,Y -560.870,Z 1255.687,A 0.000,B 0.000,C 90.000,E1 159.699} C_DIS
LIN {X -0.042,Y -562.673,Z 1255.684,A 0.000,B 0.000,C 90.000,E1 159.156} C_DIS
LIN {X 0.199,Y -566.933,Z 1255.678,A 0.000,B 0.000,C 90.000,E1 158.028} C_DIS
LIN {X 0.297,Y -571.773,Z 1255.672,A 0.000,B 0.000,C 90.000,E1 156.922} C_DIS
LIN {X -0.141,Y -578.005,Z 1255.665,A 0.000,B 0.000,C 90.000,E1 155.741} C_DIS
LIN {X 0.150,Y -586.248,Z 1255.657,A 0.000,B 0.000,C 90.000,E1 154.229} C_DIS
LIN {X 0.064,Y -590.895,Z 1255.652,A 0.000,B 0.000,C 90.000,E1 153.435} C_DIS
LIN {X 0.249,Y -596.185,Z 1255.647,A 0.000,B 0.000,C 90.000,E1 152.487} C_DIS
LIN {X 0.070,Y -599.861,Z 1255.644,A 0.000,B 0.000,C 90.000,E1 151.847} C_DIS
LIN {X 0.108,Y -604.916,Z 1255.639,A 0.000,B 0.000,C 90.000,E1 150.923} C_DIS
LIN {X 0.210,Y -609.702,Z 1255.634,A 0.000,B 0.000,C 90.000,E1 149.999} C_DIS
LIN {X 0.140,Y -611.755,Z 1255.631,A 0.000,B 0.000,C 90.000,E1 149.616} C_DIS
LIN {X -0.157,Y -614.418,Z 1255.628,A 0.000,B 0.000,C 90.000,E1 149.125} C_DIS
LIN {X 0.057,Y -619.077,Z 1255.623,A 0.000,B 0.000,C 90.000,E1 148.201} C_DIS
LIN {X 0.113,Y -625.403,Z 1255.616,A 0.000,B 0.000,C 90.000,E1 146.914} C_DIS
LIN {X -0.084,Y -628.953,Z 1255.612,A 0.000,B 0.000,C 90.000,E1 146.167} C_DIS
LIN {X 0.100,Y -632.364,Z 1255.608,A 0.000,B 0.000,C 90.000,E1 145.388} C_DIS
LIN {X -0.182,Y -636.471,Z 1255.602,A 0.000,B 0.000,C 90.000,E1 144.402} C_DIS
LIN {X 0.087,Y -639.357,Z 1255.598,A 0.000,B 0.000,C 90.000,E1 143.623} C_DIS
LIN {X 0.387,Y -642.002,Z 1255.594,A 0.000,B 0.000,C 90.000,E1 142.844} C_DIS
LIN {X -0.288,Y -645.284,Z 1255.588,A 0.000,B 0.000,C 90.000,E1 141.904} C_DIS
LIN {X -0.019,Y -648.270,Z 1255.583,A 0.000,B 0.000,C 90.000,E1 140.884} C_DIS
LIN {X 0.165,Y -652.422,Z 1255.574,A 0.000,B 0.000,C 90.000,E1 139.380} C_DIS
LIN {X 0.027,Y -655.130,Z 1255.569,A 0.000,B 0.000,C 90.000,E1 138.405} C_DIS
LIN {X 0.326,Y -658.384,Z 1255.562,A 0.000,B 0.000,C 90.000,E1 137.148} C_DIS
LIN {X -0.311,Y -664.055,Z 1255.550,A 0.000,B 0.000,C 90.000,E1 135.000} C_DIS
LIN {X 0.150,Y -668.808,Z 1255.540,A 0.000,B 0.000,C 90.000,E1 133.257} C_DIS
LIN {X -0.248,Y -672.900,Z 1255.532,A 0.000,B 0.000,C 90.000,E1 131.838} C_DIS
LIN {X -0.077,Y -676.856,Z 1255.524,A 0.000,B 0.000,C 90.000,E1 130.378} C_DIS
LIN {X -0.304,Y -680.068,Z 1255.518,A 0.000,B 0.000,C 90.000,E1 129.197} C_DIS
LIN {X 0.089,Y -683.775,Z 1255.510,A 0.000,B 0.000,C 90.000,E1 127.729} C_DIS
LIN {X 0.104,Y -686.891,Z 1255.503,A 0.000,B 0.000,C 90.000,E1 126.537} C_DIS
LIN {X 0.018,Y -689.750,Z 1255.496,A 0.000,B 0.000,C 90.000,E1 125.358} C_DIS
LIN {X 0.092,Y -691.857,Z 1255.491,A 0.000,B 0.000,C 90.000,E1 124.405} C_DIS
LIN {X 0.205,Y -693.860,Z 1255.486,A 0.000,B 0.000,C 90.000,E1 123.452} C_DIS
LIN {X 0.001,Y -696.251,Z 1255.479,A 0.000,B 0.000,C 90.000,E1 122.291} C_DIS
LIN {X -0.172,Y -698.512,Z 1255.473,A 0.000,B 0.000,C 90.000,E1 121.131} C_DIS
LIN {X -0.338,Y -700.135,Z 1255.468,A 0.000,B 0.000,C 90.000,E1 120.207} C_DIS
LIN {X -0.139,Y -701.627,Z 1255.463,A 0.000,B 0.000,C 90.000,E1 119.255} C_DIS
LIN {X -0.331,Y -703.187,Z 1255.456,A 0.000,B 0.000,C 90.000,E1 118.103} C_DIS
LIN {X 0.176,Y -704.140,Z 1255.451,A 0.000,B 0.000,C 90.000,E1 117.129} C_DIS
LIN {X 0.119,Y -704.441,Z 1255.448,A 0.000,B 0.000,C 90.000,E1 116.668} C_DIS
LIN {X 0.035,Y -704.729,Z 1255.444,A 0.000,B 0.000,C 90.000,E1 115.976} C_DIS
LIN {X 0.322,Y -704.788,Z 1255.443,A 0.000,B 0.000,C 90.000,E1 115.720} C_DIS
LIN {X 0.247,Y -704.521,Z 1255.439,A 0.000,B 0.000,C 90.000,E1 115.027} C_DIS
LIN {X -0.116,Y -704.157,Z 1255.437,A 0.000,B 0.000,C 90.000,E1 114.591} C_DIS
LIN {X -0.189,Y -703.329,Z 1255.434,A 0.000,B 0.000,C 90.000,E1 114.131} C_DIS
LIN {X -0.194,Y -702.634,Z 1255.433,A 0.000,B 0.000,C 90.000,E1 113.898} C_DIS
LIN {X 0.361,Y -700.700,Z 1255.430,A 0.000,B 0.000,C 90.000,E1 113.387} C_DIS
LIN {X -0.424,Y -699.985,Z 1255.429,A 0.000,B 0.000,C 90.000,E1 113.334} C_DIS
LIN {X 0.106,Y -695.797,Z 1255.427,A 0.000,B 0.000,C 90.000,E1 112.823} C_DIS
LIN {X -0.035,Y -694.516,Z 1255.426,A 0.000,B 0.000,C 90.000,E1 112.717} C_DIS
LIN {X 0.145,Y -692.570,Z 1255.426,A 0.000,B 0.000,C 90.000,E1 112.589} C_DIS
LIN {X 0.190,Y -687.815,Z 1255.425,A 0.000,B 0.000,C 90.000,E1 112.408} C_DIS
LIN {X 0.319,Y -685.524,Z 1255.424,A 0.000,B 0.000,C 90.000,E1 112.333} C_DIS
LIN {X 0.377,Y -677.450,Z 1255.424,A 0.000,B 0.000,C 90.000,E1 112.206} C_DIS
LIN {X 0.338,Y -676.981,Z 1255.424,A 0.000,B 0.000,C 90.000,E1 112.206} C_DIS
LIN {X 0.297,Y -670.719,Z 1255.424,A 0.000,B 0.000,C 90.000,E1 112.206} C_DIS
LIN {X 0.221,Y -629.602,Z 1255.424,A 0.000,B 0.000,C 90.000,E1 112.206} C_DIS
LIN {X -0.308,Y -627.006,Z 1255.423,A 0.000,B 0.000,C 90.000,E1 112.153} C_DIS
LIN {X -0.197,Y -625.633,Z 1255.422,A 0.000,B 0.000,C 90.000,E1 112.025} C_DIS
LIN {X -0.236,Y -625.601,Z 1255.422,A 0.000,B 0.000,C 90.000,E1 112.025} C_DIS
LIN {X 0.221,Y -625.395,Z 1255.422,A 0.000,B 0.000,C 90.000,E1 111.897} C_DIS
LIN {X 0.182,Y -625.397,Z 1255.422,A 0.000,B 0.000,C 90.000,E1 111.897} C_DIS
LIN {X 0.063,Y -626.451,Z 1255.420,A 0.000,B 0.000,C 90.000,E1 111.589} C_DIS
LIN {X -0.127,Y -628.312,Z 1255.418,A 0.000,B 0.000,C 90.000,E1 111.227} C_DIS
LIN {X 0.272,Y -632.983,Z 1255.414,A 0.000,B 0.000,C 90.000,E1 110.429} C_DIS
LIN {X 0.096,Y -636.015,Z 1255.411,A 0.000,B 0.000,C 90.000,E1 109.939} C_DIS
LIN {X -0.242,Y -640.006,Z 1255.407,A 0.000,B 0.000,C 90.000,E1 109.214} C_DIS
LIN {X 0.133,Y -645.460,Z 1255.400,A 0.000,B 0.000,C 90.000,E1 108.055} C_DIS
LIN {X 0.222,Y -651.376,Z 1255.394,A 0.000,B 0.000,C 90.000,E1 106.804} C_DIS
LIN {X 0.022,Y -654.655,Z 1255.389,A 0.000,B 0.000,C 90.000,E1 106.079} C_DIS
LIN {X -0.217,Y -656.641,Z 1255.387,A 0.000,B 0.000,C 90.000,E1 105.607} C_DIS
LIN {X 0.257,Y -659.163,Z 1255.383,A 0.000,B 0.000,C 90.000,E1 104.828} C_DIS
LIN {X -0.052,Y -661.207,Z 1255.378,A 0.000,B 0.000,C 90.000,E1 104.120} C_DIS
LIN {X 0.303,Y -662.629,Z 1255.374,A 0.000,B 0.000,C 90.000,E1 103.355} C_DIS
LIN {X 0.118,Y -663.301,Z 1255.372,A 0.000,B 0.000,C 90.000,E1 102.883} C_DIS
LIN {X -0.065,Y -663.703,Z 1255.369,A 0.000,B 0.000,C 90.000,E1 102.411} C_DIS
LIN {X 0.177,Y -663.787,Z 1255.365,A 0.000,B 0.000,C 90.000,E1 101.658} C_DIS
LIN {X -0.003,Y -663.443,Z 1255.362,A 0.000,B 0.000,C 90.000,E1 101.186} C_DIS
LIN {X -0.189,Y -662.902,Z 1255.359,A 0.000,B 0.000,C 90.000,E1 100.715} C_DIS
LIN {X 0.151,Y -662.045,Z 1255.357,A 0.000,B 0.000,C 90.000,E1 100.197} C_DIS
LIN {X 0.053,Y -661.541,Z 1255.355,A 0.000,B 0.000,C 90.000,E1 99.962} C_DIS
LIN {X -0.260,Y -660.317,Z 1255.353,A 0.000,B 0.000,C 90.000,E1 99.500} C_DIS
LIN {X 0.176,Y -658.682,Z 1255.350,A 0.000,B 0.000,C 90.000,E1 98.973} C_DIS
LIN {X -0.151,Y -656.672,Z 1255.347,A 0.000,B 0.000,C 90.000,E1 98.511} C_DIS
LIN {X 0.161,Y -654.322,Z 1255.344,A 0.000,B 0.000,C 90.000,E1 97.992} C_DIS
LIN {X -0.189,Y -651.650,Z 1255.342,A 0.000,B 0.000,C 90.000,E1 97.530} C_DIS
LIN {X 0.202,Y -649.436,Z 1255.340,A 0.000,B 0.000,C 90.000,E1 97.125} C_DIS
LIN {X -0.180,Y -646.134,Z 1255.337,A 0.000,B 0.000,C 90.000,E1 96.663} C_DIS
LIN {X 0.059,Y -642.446,Z 1255.334,A 0.000,B 0.000,C 90.000,E1 96.144} C_DIS
LIN {X 0.270,Y -638.468,Z 1255.331,A 0.000,B 0.000,C 90.000,E1 95.625} C_DIS
LIN {X -0.310,Y -632.716,Z 1255.328,A 0.000,B 0.000,C 90.000,E1 95.049} C_DIS
LIN {X -0.085,Y -627.682,Z 1255.325,A 0.000,B 0.000,C 90.000,E1 94.531} C_DIS
LIN {X 0.282,Y -622.432,Z 1255.323,A 0.000,B 0.000,C 90.000,E1 94.012} C_DIS
LIN {X 0.251,Y -615.646,Z 1255.319,A 0.000,B 0.000,C 90.000,E1 93.440} C_DIS
LIN {X -0.179,Y -609.858,Z 1255.317,A 0.000,B 0.000,C 90.000,E1 93.037} C_DIS
LIN {X -0.221,Y -602.316,Z 1255.314,A 0.000,B 0.000,C 90.000,E1 92.522} C_DIS
LIN {X -0.197,Y -596.143,Z 1255.312,A 0.000,B 0.000,C 90.000,E1 92.121} C_DIS
LIN {X 0.009,Y -589.554,Z 1255.310,A 0.000,B 0.000,C 90.000,E1 91.718} C_DIS
LIN {X 0.022,Y -582.531,Z 1255.308,A 0.000,B 0.000,C 90.000,E1 91.375} C_DIS
LIN {X -0.015,Y -574.957,Z 1255.306,A 0.000,B 0.000,C 90.000,E1 91.088} C_DIS
LIN {X -0.168,Y -571.841,Z 1255.305,A 0.000,B 0.000,C 90.000,E1 90.974} C_DIS
LIN {X -0.283,Y -570.643,Z 1255.305,A 0.000,B 0.000,C 90.000,E1 90.917} C_DIS
LIN {X 0.202,Y -568.290,Z 1255.304,A 0.000,B 0.000,C 90.000,E1 90.688} C_DIS
LIN {X 0.167,Y -568.251,Z 1255.304,A 0.000,B 0.000,C 90.000,E1 90.688} C_DIS
LIN {X 0.121,Y -567.540,Z 1255.303,A 0.000,B 0.000,C 90.000,E1 90.516} C_DIS
LIN {X -0.091,Y -567.250,Z 1255.300,A 0.000,B 0.000,C 90.000,E1 90.057} C_DIS
LIN {X -0.279,Y -569.336,Z 1255.284,A 0.000,B 0.000,C 90.000,E1 87.135} C_DIS
LIN {X -0.191,Y -571.622,Z 1255.270,A 0.000,B 0.000,C 90.000,E1 84.666} C_DIS
LIN {X 0.148,Y -573.339,Z 1255.261,A 0.000,B 0.000,C 90.000,E1 82.996} C_DIS
LIN {X 0.025,Y -575.086,Z 1255.252,A 0.000,B 0.000,C 90.000,E1 81.376} C_DIS
LIN {X -0.178,Y -576.431,Z 1255.245,A 0.000,B 0.000,C 90.000,E1 80.038} C_DIS
LIN {X 0.104,Y -577.308,Z 1255.239,A 0.000,B 0.000,C 90.000,E1 78.926} C_DIS
LIN {X 0.151,Y -578.564,Z 1255.230,A 0.000,B 0.000,C 90.000,E1 77.297} C_DIS
LIN {X 0.125,Y -579.839,Z 1255.219,A 0.000,B 0.000,C 90.000,E1 75.408} C_DIS
LIN {X 0.066,Y -580.810,Z 1255.210,A 0.000,B 0.000,C 90.000,E1 73.795} C_DIS
LIN {X 0.080,Y -582.106,Z 1255.198,A 0.000,B 0.000,C 90.000,E1 71.638} C_DIS
LIN {X 0.040,Y -582.908,Z 1255.191,A 0.000,B 0.000,C 90.000,E1 70.296} C_DIS
LIN {X 0.346,Y -584.371,Z 1255.177,A 0.000,B 0.000,C 90.000,E1 67.847} C_DIS
LIN {X -0.177,Y -586.251,Z 1255.164,A 0.000,B 0.000,C 90.000,E1 65.485} C_DIS
LIN {X 0.059,Y -587.805,Z 1255.153,A 0.000,B 0.000,C 90.000,E1 63.589} C_DIS
LIN {X 0.237,Y -589.809,Z 1255.141,A 0.000,B 0.000,C 90.000,E1 61.435} C_DIS
LIN {X -0.119,Y -591.490,Z 1255.133,A 0.000,B 0.000,C 90.000,E1 59.871} C_DIS
LIN {X 0.155,Y -593.133,Z 1255.124,A 0.000,B 0.000,C 90.000,E1 58.250} C_DIS
LIN {X 0.253,Y -594.453,Z 1255.116,A 0.000,B 0.000,C 90.000,E1 56.914} C_DIS
LIN {X 0.080,Y -595.948,Z 1255.108,A 0.000,B 0.000,C 90.000,E1 55.341} C_DIS
LIN {X -0.095,Y -597.131,Z 1255.100,A 0.000,B 0.000,C 90.000,E1 54.036} C_DIS
LIN {X 0.118,Y -598.447,Z 1255.091,A 0.000,B 0.000,C 90.000,E1 52.431} C_DIS
LIN {X 0.127,Y -599.280,Z 1255.086,A 0.000,B 0.000,C 90.000,E1 51.376} C_DIS
LIN {X -0.221,Y -599.989,Z 1255.080,A 0.000,B 0.000,C 90.000,E1 50.356} C_DIS
LIN {X -0.180,Y -600.431,Z 1255.074,A 0.000,B 0.000,C 90.000,E1 49.299} C_DIS
LIN {X -0.133,Y -600.963,Z 1255.068,A 0.000,B 0.000,C 90.000,E1 48.243} C_DIS
LIN {X 0.114,Y -601.349,Z 1255.061,A 0.000,B 0.000,C 90.000,E1 46.905} C_DIS
LIN {X -0.052,Y -601.713,Z 1255.053,A 0.000,B 0.000,C 90.000,E1 45.607} C_DIS
LIN {X -0.027,Y -601.695,Z 1255.048,A 0.000,B 0.000,C 90.000,E1 44.555} C_DIS
LIN {X 0.223,Y -601.452,Z 1255.040,A 0.000,B 0.000,C 90.000,E1 43.218} C_DIS
LIN {X 0.066,Y -600.972,Z 1255.033,A 0.000,B 0.000,C 90.000,E1 41.919} C_DIS
LIN {X 0.121,Y -600.614,Z 1255.027,A 0.000,B 0.000,C 90.000,E1 40.862} C_DIS
LIN {X -0.050,Y -599.818,Z 1255.020,A 0.000,B 0.000,C 90.000,E1 39.564} C_DIS
LIN {X -0.021,Y -599.139,Z 1255.014,A 0.000,B 0.000,C 90.000,E1 38.508} C_DIS
LIN {X -0.144,Y -598.468,Z 1255.010,A 0.000,B 0.000,C 90.000,E1 37.729} C_DIS
LIN {X -0.268,Y -597.685,Z 1255.005,A 0.000,B 0.000,C 90.000,E1 36.950} C_DIS
LIN {X 0.069,Y -595.970,Z 1254.998,A 0.000,B 0.000,C 90.000,E1 35.598} C_DIS
LIN {X 0.144,Y -594.326,Z 1254.992,A 0.000,B 0.000,C 90.000,E1 34.532} C_DIS
LIN {X 0.066,Y -591.763,Z 1254.985,A 0.000,B 0.000,C 90.000,E1 33.214} C_DIS
LIN {X 0.040,Y -589.838,Z 1254.980,A 0.000,B 0.000,C 90.000,E1 32.418} C_DIS
LIN {X 0.189,Y -586.830,Z 1254.974,A 0.000,B 0.000,C 90.000,E1 31.337} C_DIS
LIN {X 0.121,Y -584.133,Z 1254.970,A 0.000,B 0.000,C 90.000,E1 30.541} C_DIS
LIN {X 0.027,Y -580.994,Z 1254.965,A 0.000,B 0.000,C 90.000,E1 29.745} C_DIS
LIN {X 0.040,Y -578.681,Z 1254.962,A 0.000,B 0.000,C 90.000,E1 29.205} C_DIS
LIN {X -0.118,Y -574.852,Z 1254.958,A 0.000,B 0.000,C 90.000,E1 28.409} C_DIS
LIN {X -0.005,Y -571.358,Z 1254.954,A 0.000,B 0.000,C 90.000,E1 27.719} C_DIS
LIN {X -0.161,Y -567.477,Z 1254.950,A 0.000,B 0.000,C 90.000,E1 27.052} C_DIS
LIN {X -0.012,Y -564.126,Z 1254.947,A 0.000,B 0.000,C 90.000,E1 26.488} C_DIS
LIN {X -0.081,Y -558.688,Z 1254.943,A 0.000,B 0.000,C 90.000,E1 25.668} C_DIS
LIN {X 0.138,Y -553.764,Z 1254.939,A 0.000,B 0.000,C 90.000,E1 24.951} C_DIS
LIN {X -0.044,Y -547.238,Z 1254.934,A 0.000,B 0.000,C 90.000,E1 24.131} C_DIS
LIN {X 0.333,Y -541.433,Z 1254.930,A 0.000,B 0.000,C 90.000,E1 23.387} C_DIS
LIN {X -0.288,Y -532.567,Z 1254.925,A 0.000,B 0.000,C 90.000,E1 22.461} C_DIS
LIN {X 0.108,Y -526.004,Z 1254.921,A 0.000,B 0.000,C 90.000,E1 21.716} C_DIS
LIN {X -0.087,Y -516.920,Z 1254.916,A 0.000,B 0.000,C 90.000,E1 20.791} C_DIS
LIN {X -0.278,Y -506.491,Z 1254.910,A 0.000,B 0.000,C 90.000,E1 19.758} C_DIS
LIN {X -0.044,Y -495.207,Z 1254.904,A 0.000,B 0.000,C 90.000,E1 18.652} C_DIS
LIN {X -0.147,Y -485.359,Z 1254.899,A 0.000,B 0.000,C 90.000,E1 17.764} C_DIS
LIN {X 0.015,Y -478.211,Z 1254.895,A 0.000,B 0.000,C 90.000,E1 17.094} C_DIS
LIN {X -0.086,Y -461.876,Z 1254.887,A 0.000,B 0.000,C 90.000,E1 15.662} C_DIS
LIN {X 0.167,Y -444.144,Z 1254.878,A 0.000,B 0.000,C 90.000,E1 14.008} C_DIS
LIN {X 0.027,Y -421.006,Z 1254.865,A 0.000,B 0.000,C 90.000,E1 11.715} C_DIS
LIN {X 0.091,Y -406.725,Z 1254.856,A 0.000,B 0.000,C 90.000,E1 10.141} C_DIS
LIN {X -0.193,Y -401.181,Z 1254.853,A 0.000,B 0.000,C 90.000,E1 9.557} C_DIS
LIN {X 0.129,Y -396.641,Z 1254.850,A 0.000,B 0.000,C 90.000,E1 8.916} C_DIS
LIN {X 0.146,Y -394.653,Z 1254.848,A 0.000,B 0.000,C 90.000,E1 8.568} C_DIS
LIN {X 0.108,Y -394.633,Z 1254.848,A 0.000,B 0.000,C 90.000,E1 8.568} C_DIS
LIN {X -0.184,Y -394.493,Z 1254.847,A 0.000,B 0.000,C 90.000,E1 8.511} C_DIS
LIN {X 0.168,Y -394.514,Z 1254.847,A 0.000,B 0.000,C 90.000,E1 8.454} C_DIS
LIN {X -0.132,Y -396.250,Z 1254.845,A 0.000,B 0.000,C 90.000,E1 8.106} C_DIS
LIN {X 0.106,Y -398.660,Z 1254.844,A 0.000,B 0.000,C 90.000,E1 7.814} C_DIS
LIN {X -0.168,Y -400.303,Z 1254.843,A 0.000,B 0.000,C 90.000,E1 7.701} C_DIS
LIN {X -0.182,Y -407.537,Z 1254.840,A 0.000,B 0.000,C 90.000,E1 7.182} C_DIS
LIN {X -0.014,Y -414.078,Z 1254.837,A 0.000,B 0.000,C 90.000,E1 6.720} C_DIS
LIN {X 0.056,Y -419.004,Z 1254.835,A 0.000,B 0.000,C 90.000,E1 6.372} C_DIS
LIN {X 0.040,Y -426.930,Z 1254.832,A 0.000,B 0.000,C 90.000,E1 5.796} C_DIS
LIN {X -0.088,Y -433.239,Z 1254.830,A 0.000,B 0.000,C 90.000,E1 5.334} C_DIS
LIN {X -0.006,Y -441.081,Z 1254.826,A 0.000,B 0.000,C 90.000,E1 4.702} C_DIS
LIN {X 0.213,Y -453.518,Z 1254.821,A 0.000,B 0.000,C 90.000,E1 3.669} C_DIS
LIN {X 0.182,Y -461.090,Z 1254.817,A 0.000,B 0.000,C 90.000,E1 3.037} C_DIS
LIN {X 0.062,Y -468.396,Z 1254.813,A 0.000,B 0.000,C 90.000,E1 2.407} C_DIS
LIN {X 0.059,Y -472.736,Z 1254.811,A 0.000,B 0.000,C 90.000,E1 2.007} C_DIS
LIN {X 0.002,Y -479.628,Z 1254.807,A 0.000,B 0.000,C 90.000,E1 1.318} C_DIS
LIN {X -0.095,Y -486.077,Z 1254.803,A 0.000,B 0.000,C 90.000,E1 0.630} C_DIS
LIN {X 0.000,Y -491.312,Z 1254.800,A 0.000,B 0.000,C 90.000,E1 360.000} C_DIS
LIN {X 0.078,Y -495.461,Z 1254.797,A 0.000,B 0.000,C 90.000,E1 359.484} C_DIS
LIN {X -0.018,Y -501.005,Z 1254.793,A 0.000,B 0.000,C 90.000,E1 358.740} C_DIS
LIN {X 0.150,Y -507.136,Z 1254.788,A 0.000,B 0.000,C 90.000,E1 357.822} C_DIS
LIN {X -0.052,Y -511.013,Z 1254.785,A 0.000,B 0.000,C 90.000,E1 357.249} C_DIS
LIN {X 0.233,Y -516.407,Z 1254.780,A 0.000,B 0.000,C 90.000,E1 356.331} C_DIS
LIN {X -0.100,Y -518.961,Z 1254.777,A 0.000,B 0.000,C 90.000,E1 355.927} C_DIS
LIN {X 0.047,Y -522.843,Z 1254.773,A 0.000,B 0.000,C 90.000,E1 355.179} C_DIS
LIN {X 0.229,Y -526.459,Z 1254.769,A 0.000,B 0.000,C 90.000,E1 354.432} C_DIS
LIN {X -0.084,Y -529.812,Z 1254.765,A 0.000,B 0.000,C 90.000,E1 353.742} C_DIS
LIN {X 0.187,Y -531.724,Z 1254.763,A 0.000,B 0.000,C 90.000,E1 353.280} C_DIS
LIN {X 0.231,Y -535.102,Z 1254.758,A 0.000,B 0.000,C 90.000,E1 352.413} C_DIS
LIN {X -0.162,Y -539.251,Z 1254.752,A 0.000,B 0.000,C 90.000,E1 351.310} C_DIS
LIN {X -0.113,Y -541.181,Z 1254.749,A 0.000,B 0.000,C 90.000,E1 350.735} C_DIS
LIN {X 0.118,Y -543.723,Z 1254.744,A 0.000,B 0.000,C 90.000,E1 349.859} C_DIS
LIN {X -0.165,Y -546.887,Z 1254.738,A 0.000,B 0.000,C 90.000,E1 348.757} C_DIS
LIN {X 0.233,Y -549.630,Z 1254.731,A 0.000,B 0.000,C 90.000,E1 347.589} C_DIS
LIN {X -0.165,Y -552.766,Z 1254.723,A 0.000,B 0.000,C 90.000,E1 346.228} C_DIS
LIN {X 0.188,Y -554.352,Z 1254.719,A 0.000,B 0.000,C 90.000,E1 345.353} C_DIS
LIN {X -0.106,Y -556.253,Z 1254.713,A 0.000,B 0.000,C 90.000,E1 344.267} C_DIS
LIN {X 0.017,Y -557.926,Z 1254.706,A 0.000,B 0.000,C 90.000,E1 343.142} C_DIS
LIN {X -0.213,Y -559.274,Z 1254.700,A 0.000,B 0.000,C 90.000,E1 342.054} C_DIS
LIN {X -0.194,Y -560.077,Z 1254.696,A 0.000,B 0.000,C 90.000,E1 341.221} C_DIS
LIN {X -0.210,Y -560.672,Z 1254.689,A 0.000,B 0.000,C 90.000,E1 340.115} C_DIS
LIN {X 0.218,Y -560.823,Z 1254.686,A 0.000,B 0.000,C 90.000,E1 339.518} C_DIS
LIN {X 0.316,Y -560.843,Z 1254.683,A 0.000,B 0.000,C 90.000,E1 338.954} C_DIS
LIN {X 0.006,Y -560.544,Z 1254.679,A 0.000,B 0.000,C 90.000,E1 338.156} C_DIS
LIN {X -0.102,Y -560.227,Z 1254.676,A 0.000,B 0.000,C 90.000,E1 337.614} C_DIS
LIN {X -0.208,Y -559.396,Z 1254.671,A 0.000,B 0.000,C 90.000,E1 336.794} C_DIS
LIN {X -0.110,Y -558.710,Z 1254.668,A 0.000,B 0.000,C 90.000,E1 336.230} C_DIS
LIN {X 0.283,Y -557.429,Z 1254.663,A 0.000,B 0.000,C 90.000,E1 335.357} C_DIS
LIN {X -0.138,Y -556.347,Z 1254.660,A 0.000,B 0.000,C 90.000,E1 334.845} C_DIS
LIN {X 0.000,Y -553.942,Z 1254.654,A 0.000,B 0.000,C 90.000,E1 333.717} C_DIS
LIN {X 0.076,Y -551.632,Z 1254.649,A 0.000,B 0.000,C 90.000,E1 332.871} C_DIS
LIN {X 0.132,Y -548.867,Z 1254.645,A 0.000,B 0.000,C 90.000,E1 332.025} C_DIS
LIN {X 0.158,Y -545.608,Z 1254.640,A 0.000,B 0.000,C 90.000,E1 331.179} C_DIS
LIN {X 0.273,Y -542.433,Z 1254.636,A 0.000,B 0.000,C 90.000,E1 330.461} C_DIS
LIN {X -0.114,Y -538.743,Z 1254.632,A 0.000,B 0.000,C 90.000,E1 329.793} C_DIS
LIN {X 0.074,Y -535.482,Z 1254.629,A 0.000,B 0.000,C 90.000,E1 329.203} C_DIS
LIN {X 0.034,Y -527.098,Z 1254.622,A 0.000,B 0.000,C 90.000,E1 327.916} C_DIS
LIN {X 0.057,Y -515.571,Z 1254.612,A 0.000,B 0.000,C 90.000,E1 326.167} C_DIS
LIN {X -0.269,Y -511.440,Z 1254.608,A 0.000,B 0.000,C 90.000,E1 325.468} C_DIS
LIN {X 0.170,Y -509.219,Z 1254.606,A 0.000,B 0.000,C 90.000,E1 324.975} C_DIS
LIN {X -0.112,Y -507.433,Z 1254.603,A 0.000,B 0.000,C 90.000,E1 324.562} C_DIS
LIN {X 0.304,Y -504.949,Z 1254.598,A 0.000,B 0.000,C 90.000,E1 323.623} C_DIS
LIN {X 0.066,Y -503.514,Z 1254.593,A 0.000,B 0.000,C 90.000,E1 322.763} C_DIS
LIN {X -0.265,Y -502.948,Z 1254.588,A 0.000,B 0.000,C 90.000,E1 321.904} C_DIS
LIN {X 0.132,Y -503.338,Z 1254.570,A 0.000,B 0.000,C 90.000,E1 318.566} C_DIS
LIN {X 0.036,Y -503.843,Z 1254.560,A 0.000,B 0.000,C 90.000,E1 316.782} C_DIS
LIN {X -0.284,Y -504.187,Z 1254.552,A 0.000,B 0.000,C 90.000,E1 315.324} C_DIS
LIN {X -0.007,Y -504.598,Z 1254.542,A 0.000,B 0.000,C 90.000,E1 313.500} C_DIS
LIN {X 0.162,Y -505.137,Z 1254.530,A 0.000,B 0.000,C 90.000,E1 311.391} C_DIS
LIN {X -0.223,Y -505.466,Z 1254.520,A 0.000,B 0.000,C 90.000,E1 309.644} C_DIS
LIN {X 0.073,Y -505.931,Z 1254.509,A 0.000,B 0.000,C 90.000,E1 307.523} C_DIS
LIN {X 0.272,Y -506.343,Z 1254.500,A 0.000,B 0.000,C 90.000,E1 306.011} C_DIS
LIN {X 0.175,Y -506.548,Z 1254.492,A 0.000,B 0.000,C 90.000,E1 304.532} C_DIS
LIN {X -0.207,Y -506.581,Z 1254.484,A 0.000,B 0.000,C 90.000,E1 303.086} C_DIS
LIN {X 0.155,Y -506.620,Z 1254.474,A 0.000,B 0.000,C 90.000,E1 301.258} C_DIS
LIN {X -0.118,Y -506.504,Z 1254.462,A 0.000,B 0.000,C 90.000,E1 299.205} C_DIS
LIN {X 0.224,Y -506.413,Z 1254.456,A 0.000,B 0.000,C 90.000,E1 297.975} C_DIS
LIN {X -0.169,Y -506.169,Z 1254.446,A 0.000,B 0.000,C 90.000,E1 296.232} C_DIS
LIN {X 0.032,Y -506.162,Z 1254.437,A 0.000,B 0.000,C 90.000,E1 294.719} C_DIS
LIN {X 0.236,Y -506.121,Z 1254.429,A 0.000,B 0.000,C 90.000,E1 293.206} C_DIS
LIN {X 0.233,Y -505.762,Z 1254.421,A 0.000,B 0.000,C 90.000,E1 291.716} C_DIS
LIN {X 0.036,Y -505.091,Z 1254.413,A 0.000,B 0.000,C 90.000,E1 290.248} C_DIS
LIN {X -0.167,Y -503.915,Z 1254.398,A 0.000,B 0.000,C 90.000,E1 287.583} C_DIS
LIN {X -0.158,Y -503.422,Z 1254.391,A 0.000,B 0.000,C 90.000,E1 286.386} C_DIS
LIN {X -0.226,Y -502.706,Z 1254.383,A 0.000,B 0.000,C 90.000,E1 284.898} C_DIS
LIN {X 0.239,Y -501.917,Z 1254.376,A 0.000,B 0.000,C 90.000,E1 283.647} C_DIS
LIN {X 0.004,Y -500.764,Z 1254.368,A 0.000,B 0.000,C 90.000,E1 282.175} C_DIS
LIN {X 0.055,Y -499.212,Z 1254.358,A 0.000,B 0.000,C 90.000,E1 280.366} C_DIS
LIN {X 0.070,Y -498.068,Z 1254.349,A 0.000,B 0.000,C 90.000,E1 278.859} C_DIS
LIN {X -0.178,Y -496.567,Z 1254.338,A 0.000,B 0.000,C 90.000,E1 276.777} C_DIS
LIN {X -0.035,Y -495.388,Z 1254.326,A 0.000,B 0.000,C 90.000,E1 274.645} C_DIS
LIN {X -0.206,Y -494.494,Z 1254.317,A 0.000,B 0.000,C 90.000,E1 273.151} C_DIS
LIN {X 0.072,Y -493.514,Z 1254.309,A 0.000,B 0.000,C 90.000,E1 271.604} C_DIS
LIN {X -0.126,Y -491.937,Z 1254.296,A 0.000,B 0.000,C 90.000,E1 269.198} C_DIS
LIN {X 0.154,Y -490.599,Z 1254.282,A 0.000,B 0.000,C 90.000,E1 266.731} C_DIS
LIN {X 0.229,Y -489.749,Z 1254.272,A 0.000,B 0.000,C 90.000,E1 264.894} C_DIS
LIN {X 0.009,Y -488.867,Z 1254.263,A 0.000,B 0.000,C 90.000,E1 263.394} C_DIS
LIN {X -0.109,Y -487.981,Z 1254.257,A 0.000,B 0.000,C 90.000,E1 262.186} C_DIS
LIN {X 0.015,Y -487.095,Z 1254.251,A 0.000,B 0.000,C 90.000,E1 261.254} C_DIS
LIN {X 0.163,Y -485.380,Z 1254.241,A 0.000,B 0.000,C 90.000,E1 259.398} C_DIS
LIN {X 0.058,Y -483.360,Z 1254.226,A 0.000,B 0.000,C 90.000,E1 256.645} C_DIS
LIN {X 0.249,Y -481.835,Z 1254.212,A 0.000,B 0.000,C 90.000,E1 254.157} C_DIS
LIN {X -0.233,Y -480.827,Z 1254.202,A 0.000,B 0.000,C 90.000,E1 252.362} C_DIS
LIN {X -0.150,Y -479.678,Z 1254.190,A 0.000,B 0.000,C 90.000,E1 250.188} C_DIS
LIN {X 0.252,Y -478.828,Z 1254.181,A 0.000,B 0.000,C 90.000,E1 248.592} C_DIS
LIN {X 0.157,Y -477.732,Z 1254.169,A 0.000,B 0.000,C 90.000,E1 246.433} C_DIS
LIN {X -0.158,Y -476.814,Z 1254.162,A 0.000,B 0.000,C 90.000,E1 245.229} C_DIS
LIN {X -0.054,Y -476.040,Z 1254.155,A 0.000,B 0.000,C 90.000,E1 243.973} C_DIS
LIN {X -0.037,Y -474.770,Z 1254.145,A 0.000,B 0.000,C 90.000,E1 242.103} C_DIS
LIN {X 0.175,Y -473.403,Z 1254.135,A 0.000,B 0.000,C 90.000,E1 240.205} C_DIS
LIN {X -0.167,Y -472.387,Z 1254.128,A 0.000,B 0.000,C 90.000,E1 238.997} C_DIS
LIN {X 0.049,Y -471.058,Z 1254.119,A 0.000,B 0.000,C 90.000,E1 237.406} C_DIS
LIN {X 0.049,Y -469.009,Z 1254.105,A 0.000,B 0.000,C 90.000,E1 234.895} C_DIS
LIN {X 0.084,Y -467.059,Z 1254.088,A 0.000,B 0.000,C 90.000,E1 231.743} C_DIS
LIN {X 0.267,Y -466.127,Z 1254.077,A 0.000,B 0.000,C 90.000,E1 229.828} C_DIS
LIN {X -0.037,Y -465.297,Z 1254.068,A 0.000,B 0.000,C 90.000,E1 228.286} C_DIS
LIN {X 0.182,Y -464.757,Z 1254.063,A 0.000,B 0.000,C 90.000,E1 227.310} C_DIS
LIN {X 0.225,Y -463.672,Z 1254.052,A 0.000,B 0.000,C 90.000,E1 225.405} C_DIS
LIN {X -0.016,Y -462.206,Z 1254.030,A 0.000,B 0.000,C 90.000,E1 221.310} C_DIS
LIN {X 0.064,Y -463.533,Z 1254.003,A 0.000,B 0.000,C 90.000,E1 216.537} C_DIS
LIN {X -0.153,Y -466.747,Z 1253.979,A 0.000,B 0.000,C 90.000,E1 212.133} C_DIS
LIN {X -0.121,Y -469.054,Z 1253.966,A 0.000,B 0.000,C 90.000,E1 209.922} C_DIS
LIN {X -0.077,Y -471.790,Z 1253.954,A 0.000,B 0.000,C 90.000,E1 207.719} C_DIS
LIN {X 0.109,Y -476.150,Z 1253.935,A 0.000,B 0.000,C 90.000,E1 204.259} C_DIS
LIN {X 0.160,Y -479.468,Z 1253.923,A 0.000,B 0.000,C 90.000,E1 202.078} C_DIS
LIN {X -0.191,Y -486.123,Z 1253.902,A 0.000,B 0.000,C 90.000,E1 198.417} C_DIS
LIN {X 0.021,Y -488.662,Z 1253.895,A 0.000,B 0.000,C 90.000,E1 197.166} C_DIS
LIN {X -0.170,Y -491.906,Z 1253.887,A 0.000,B 0.000,C 90.000,E1 195.662} C_DIS
LIN {X -0.064,Y -495.854,Z 1253.877,A 0.000,B 0.000,C 90.000,E1 193.828} C_DIS
LIN {X -0.059,Y -500.553,Z 1253.865,A 0.000,B 0.000,C 90.000,E1 191.715} C_DIS
LIN {X 0.028,Y -504.784,Z 1253.855,A 0.000,B 0.000,C 90.000,E1 189.905} C_DIS
LIN {X -0.279,Y -507.595,Z 1253.849,A 0.000,B 0.000,C 90.000,E1 188.746} C_DIS
LIN {X -0.084,Y -511.215,Z 1253.840,A 0.000,B 0.000,C 90.000,E1 187.239} C_DIS
LIN {X 0.025,Y -515.491,Z 1253.830,A 0.000,B 0.000,C 90.000,E1 185.454} C_DIS
LIN {X 0.231,Y -519.693,Z 1253.821,A 0.000,B 0.000,C 90.000,E1 183.669} C_DIS
LIN {X 0.034,Y -522.445,Z 1253.814,A 0.000,B 0.000,C 90.000,E1 182.522} C_DIS
LIN {X -0.200,Y -526.469,Z 1253.804,A 0.000,B 0.000,C 90.000,E1 180.802} C_DIS
LIN {X 0.191,Y -529.785,Z 1253.796,A 0.000,B 0.000,C 90.000,E1 179.312} C_DIS
LIN {X 0.138,Y -532.310,Z 1253.790,A 0.000,B 0.000,C 90.000,E1 178.165} C_DIS
LIN {X 0.101,Y -534.741,Z 1253.784,A 0.000,B 0.000,C 90.000,E1 177.020} C_DIS
LIN {X 0.154,Y -537.602,Z 1253.776,A 0.000,B 0.000,C 90.000,E1 175.584} C_DIS
LIN {X -0.277,Y -540.212,Z 1253.768,A 0.000,B 0.000,C 90.000,E1 174.204} C_DIS
LIN {X -0.147,Y -541.730,Z 1253.763,A 0.000,B 0.000,C 90.000,E1 173.337} C_DIS
LIN {X 0.089,Y -544.061,Z 1253.755,A 0.000,B 0.000,C 90.000,E1 171.894} C_DIS
LIN {X -0.186,Y -545.790,Z 1253.749,A 0.000,B 0.000,C 90.000,E1 170.792} C_DIS
LIN {X 0.196,Y -547.754,Z 1253.741,A 0.000,B 0.000,C 90.000,E1 169.342} C_DIS
LIN {X 0.068,Y -549.207,Z 1253.735,A 0.000,B 0.000,C 90.000,E1 168.229} C_DIS
LIN {X 0.072,Y -550.853,Z 1253.727,A 0.000,B 0.000,C 90.000,E1 166.825} C_DIS
LIN {X 0.177,Y -553.533,Z 1253.714,A 0.000,B 0.000,C 90.000,E1 164.574} C_DIS
LIN {X -0.134,Y -556.344,Z 1253.704,A 0.000,B 0.000,C 90.000,E1 162.653} C_DIS
LIN {X -0.259,Y -559.222,Z 1253.696,A 0.000,B 0.000,C 90.000,E1 161.275} C_DIS
LIN {X -0.159,Y -562.974,Z 1253.688,A 0.000,B 0.000,C 90.000,E1 159.880} C_DIS
LIN {X 0.076,Y -565.776,Z 1253.684,A 0.000,B 0.000,C 90.000,E1 159.028} C_DIS
LIN {X 0.061,Y -570.767,Z 1253.677,A 0.000,B 0.000,C 90.000,E1 157.794} C_DIS
LIN {X -0.318,Y -575.784,Z 1253.671,A 0.000,B 0.000,C 90.000,E1 156.741} C_DIS
LIN {X -0.072,Y -583.515,Z 1253.662,A 0.000,B 0.000,C 90.000,E1 155.229} C_DIS
LIN {X -0.144,Y -590.938,Z 1253.655,A 0.000,B 0.000,C 90.000,E1 153.896} C_DIS
LIN {X -0.009,Y -596.739,Z 1253.649,A 0.000,B 0.000,C 90.000,E1 152.820} C_DIS
LIN {X -0.084,Y -603.075,Z 1253.642,A 0.000,B 0.000,C 90.000,E1 151.641} C_DIS
LIN {X 0.050,Y -606.477,Z 1253.639,A 0.000,B 0.000,C 90.000,E1 150.973} C_DIS
LIN {X -0.107,Y -610.432,Z 1253.635,A 0.000,B 0.000,C 90.000,E1 150.205} C_DIS
LIN {X 0.134,Y -612.422,Z 1253.632,A 0.000,B 0.000,C 90.000,E1 149.793} C_DIS
LIN {X 0.040,Y -615.634,Z 1253.629,A 0.000,B 0.000,C 90.000,E1 149.154} C_DIS
LIN {X -0.216,Y -617.511,Z 1253.627,A 0.000,B 0.000,C 90.000,E1 148.791} C_DIS
LIN {X 0.040,Y -621.351,Z 1253.622,A 0.000,B 0.000,C 90.000,E1 147.995} C_DIS
LIN {X -0.198,Y -625.646,Z 1253.617,A 0.000,B 0.000,C 90.000,E1 147.120} C_DIS
LIN {X -0.049,Y -630.239,Z 1253.612,A 0.000,B 0.000,C 90.000,E1 146.087} C_DIS
LIN {X 0.159,Y -634.497,Z 1253.606,A 0.000,B 0.000,C 90.000,E1 145.055} C_DIS
LIN {X -0.100,Y -638.464,Z 1253.600,A 0.000,B 0.000,C 90.000,E1 144.069} C_DIS
LIN {X 0.186,Y -641.187,Z 1253.596,A 0.000,B 0.000,C 90.000,E1 143.290} C_DIS
LIN {X -0.111,Y -644.501,Z 1253.591,A 0.000,B 0.000,C 90.000,E1 142.316} C_DIS
LIN {X -0.247,Y -647.516,Z 1253.585,A 0.000,B 0.000,C 90.000,E1 141.331} C_DIS
LIN {X 0.047,Y -650.352,Z 1253.580,A 0.000,B 0.000,C 90.000,E1 140.312} C_DIS
LIN {X -0.228,Y -654.407,Z 1253.571,A 0.000,B 0.000,C 90.000,E1 138.852} C_DIS
LIN {X -0.417,Y -658.320,Z 1253.563,A 0.000,B 0.000,C 90.000,E1 137.391} C_DIS
LIN {X -0.115,Y -663.226,Z 1253.552,A 0.000,B 0.000,C 90.000,E1 135.405} C_DIS
LIN {X -0.154,Y -668.550,Z 1253.541,A 0.000,B 0.000,C 90.000,E1 133.461} C_DIS
LIN {X -0.068,Y -672.580,Z 1253.533,A 0.000,B 0.000,C 90.000,E1 132.000} C_DIS
LIN {X 0.101,Y -676.534,Z 1253.525,A 0.000,B 0.000,C 90.000,E1 130.539} C_DIS
LIN {X -0.100,Y -680.336,Z 1253.517,A 0.000,B 0.000,C 90.000,E1 129.116} C_DIS
LIN {X 0.266,Y -683.445,Z 1253.511,A 0.000,B 0.000,C 90.000,E1 127.890} C_DIS
LIN {X -0.238,Y -687.161,Z 1253.503,A 0.000,B 0.000,C 90.000,E1 126.503} C_DIS
LIN {X 0.198,Y -689.431,Z 1253.497,A 0.000,B 0.000,C 90.000,E1 125.518} C_DIS
LIN {X 0.306,Y -692.094,Z 1253.491,A 0.000,B 0.000,C 90.000,E1 124.326} C_DIS
LIN {X -0.161,Y -694.105,Z 1253.486,A 0.000,B 0.000,C 90.000,E1 123.420} C_DIS
LIN {X -0.132,Y -696.972,Z 1253.478,A 0.000,B 0.000,C 90.000,E1 122.005} C_DIS
LIN {X 0.041,Y -698.717,Z 1253.473,A 0.000,B 0.000,C 90.000,E1 121.052} C_DIS
LIN {X 0.140,Y -700.761,Z 1253.466,A 0.000,B 0.000,C 90.000,E1 119.873} C_DIS
LIN {X 0.003,Y -702.174,Z 1253.461,A 0.000,B 0.000,C 90.000,E1 118.949} C_DIS
LIN {X -0.121,Y -703.407,Z 1253.456,A 0.000,B 0.000,C 90.000,E1 118.025} C_DIS
LIN {X 0.064,Y -704.329,Z 1253.451,A 0.000,B 0.000,C 90.000,E1 117.078} C_DIS
LIN {X 0.298,Y -704.781,Z 1253.447,A 0.000,B 0.000,C 90.000,E1 116.360} C_DIS
LIN {X 0.221,Y -704.934,Z 1253.443,A 0.000,B 0.000,C 90.000,E1 115.668} C_DIS
LIN {X 0.161,Y -704.822,Z 1253.440,A 0.000,B 0.000,C 90.000,E1 115.207} C_DIS
LIN {X 0.084,Y -704.234,Z 1253.436,A 0.000,B 0.000,C 90.000,E1 114.515} C_DIS
LIN {X -0.279,Y -703.432,Z 1253.434,A 0.000,B 0.000,C 90.000,E1 114.079} C_DIS
LIN {X 0.002,Y -702.605,Z 1253.432,A 0.000,B 0.000,C 90.000,E1 113.823} C_DIS
LIN {X 0.276,Y -700.547,Z 1253.430,A 0.000,B 0.000,C 90.000,E1 113.334} C_DIS
LIN {X -0.231,Y -699.680,Z 1253.429,A 0.000,B 0.000,C 90.000,E1 113.259} C_DIS
LIN {X 0.022,Y -695.407,Z 1253.427,A 0.000,B 0.000,C 90.000,E1 112.770} C_DIS
LIN {X 0.149,Y -693.842,Z 1253.426,A 0.000,B 0.000,C 90.000,E1 112.642} C_DIS
LIN {X -0.182,Y -691.585,Z 1253.425,A 0.000,B 0.000,C 90.000,E1 112.567} C_DIS
LIN {X 0.032,Y -687.007,Z 1253.424,A 0.000,B 0.000,C 90.000,E1 112.386} C_DIS
LIN {X -0.058,Y -683.797,Z 1253.424,A 0.000,B 0.000,C 90.000,E1 112.333} C_DIS
LIN {X 0.386,Y -677.259,Z 1253.424,A 0.000,B 0.000,C 90.000,E1 112.206} C_DIS
LIN {X 0.350,Y -676.528,Z 1253.424,A 0.000,B 0.000,C 90.000,E1 112.206} C_DIS
LIN {X 0.294,Y -628.828,Z 1253.424,A 0.000,B 0.000,C 90.000,E1 112.206} C_DIS
LIN {X -0.061,Y -626.224,Z 1253.423,A 0.000,B 0.000,C 90.000,E1 112.153} C_DIS
LIN {X -0.007,Y -624.770,Z 1253.422,A 0.000,B 0.000,C 90.000,E1 112.025} C_DIS
LIN {X -0.051,Y -624.741,Z 1253.422,A 0.000,B 0.000,C 90.000,E1 112.025} C_DIS
LIN {X 0.071,Y -624.461,Z 1253.422,A 0.000,B 0.000,C 90.000,E1 111.897} C_DIS
LIN {X 0.027,Y -624.468,Z 1253.422,A 0.000,B 0.000,C 90.000,E1 111.897} C_DIS
LIN {X -0.134,Y -625.974,Z 1253.419,A 0.000,B 0.000,C 90.000,E1 111.461} C_DIS
LIN {X -0.135,Y -627.543,Z 1253.417,A 0.000,B 0.000,C 90.000,E1 111.153} C_DIS
LIN {X 0.030,Y -632.199,Z 1253.413,A 0.000,B 0.000,C 90.000,E1 110.375} C_DIS
LIN {X -0.139,Y -635.782,Z 1253.410,A 0.000,B 0.000,C 90.000,E1 109.758} C_DIS
LIN {X 0.333,Y -639.548,Z 1253.406,A 0.000,B 0.000,C 90.000,E1 108.960} C_DIS
LIN {X -0.133,Y -644.393,Z 1253.400,A 0.000,B 0.000,C 90.000,E1 108.000} C_DIS
LIN {X 0.129,Y -650.323,Z 1253.393,A 0.000,B 0.000,C 90.000,E1 106.732} C_DIS
LIN {X -0.267,Y -653.629,Z 1253.389,A 0.000,B 0.000,C 90.000,E1 106.024} C_DIS
LIN {X 0.178,Y -656.475,Z 1253.385,A 0.000,B 0.000,C 90.000,E1 105.245} C_DIS
LIN {X -0.048,Y -658.145,Z 1253.382,A 0.000,B 0.000,C 90.000,E1 104.773} C_DIS
LIN {X 0.275,Y -660.146,Z 1253.378,A 0.000,B 0.000,C 90.000,E1 104.008} C_DIS
LIN {X 0.077,Y -661.136,Z 1253.375,A 0.000,B 0.000,C 90.000,E1 103.536} C_DIS
LIN {X -0.211,Y -662.176,Z 1253.371,A 0.000,B 0.000,C 90.000,E1 102.827} C_DIS
LIN {X 0.247,Y -662.644,Z 1253.369,A 0.000,B 0.000,C 90.000,E1 102.299} C_DIS
LIN {X 0.061,Y -662.675,Z 1253.366,A 0.000,B 0.000,C 90.000,E1 101.827} C_DIS
LIN {X -0.353,Y -662.204,Z 1253.362,A 0.000,B 0.000,C 90.000,E1 101.130} C_DIS
LIN {X 0.104,Y -661.649,Z 1253.359,A 0.000,B 0.000,C 90.000,E1 100.602} C_DIS
